// TwinCAT 3 PLC project Untitled1
// ProgramVersion: 3.1.4026.19
// libraries:
//   Tc2_Standard, * (Beckhoff Automation GmbH)
//   Tc2_System, * (Beckhoff Automation GmbH)
// project tree:
//   DUTs/ eGeneralState.TcDUT, eLiftPins.TcDUT, eLiftposition.TcDUT, eLiftStates.TcDUT, eMachineStateLamp.TcDUT, eModus.TcDUT, eSchuifStates.TcDUT, eSingleState.TcDUT, eSlideposition.TcDUT, eStartStop.TcDUT, eValvePosition.TcDUT, eZuigerCilinderposition.TcDUT, eZuigerHorizontaal.TcDUT
//   / PlcTask.TcTTO
//   POUs/ FB_Band.TcPOU, FB_Blinking.TcPOU, FB_ControlSystem.TcPOU, FB_Depalletizer.TcPOU, FB_Lift.TcPOU, FB_LiftA_Extended.TcPOU, FB_LiftB_Extended.TcPOU, FB_LiftJanno.TcPOU, FB_Palletizer.TcPOU, FB_Schuif.TcPOU, FB_Zuiger.TcPOU, FB_Blinking.TcPOU, F_StateEnumToStringSingleState.TcPOU, FB_BlikjesBand.TcPOU, FB_BufferMetKlep.TcPOU, FB_BufferZonderKlep.TcPOU, FB_Invoer.TcPOU, FB_Klep.TcPOU, FB_Simulation.TcPOU, FB_StateManager.TcPOU, GVL.TcGVL, MAIN.TcPOU, F_StateEnumToStringGeneralState.TcPOU
// real-time tasks:
//   TASK PlcTask: cycle T#10ms, priority 20, ADS port 350

CONFIGURATION Untitled1
    RESOURCE PLC ON TwinCAT3
        TASK PlcTask(INTERVAL := T#10ms, PRIORITY := 20);
        PROGRAM MAIN WITH PlcTask : MAIN;
    END_RESOURCE
END_CONFIGURATION

// ---- DUTs/eGeneralState.TcDUT
{attribute 'qualified_only'}
{attribute 'strict'}
{attribute 'to_string'}
TYPE eGeneralState :
(
	Idle 		:= 0,
	Execute		:= 1,
	Stopped 	:= 2,
	Aborted 	:= 3
);
END_TYPE

// ---- DUTs/eLiftPins.TcDUT
{attribute 'qualified_only'}
{attribute 'strict'}
{attribute 'to_string'}
TYPE eLiftPins :
(
	In := 0,
	Out := 1,
	Unknown := 2
);
END_TYPE

// ---- DUTs/eLiftposition.TcDUT
{attribute 'qualified_only'}
{attribute 'strict'}
{attribute 'to_string'}
TYPE eLiftposition :
(
	Idle		:= 0,
	GoingUp 	:= 1,
	GoingDown 	:= 2
	
);
END_TYPE

// ---- DUTs/eLiftStates.TcDUT
{attribute 'qualified_only'}
{attribute 'strict'}
{attribute 'to_string'}
TYPE eLiftStates :
(
	InitHome := 0,
    MoveToHome := 1,
    Impale := 2,
    MoveUpToLayer := 3
);
END_TYPE

// ---- DUTs/eMachineStateLamp.TcDUT
{attribute 'qualified_only'}
{attribute 'strict'}
{attribute 'to_string'}
TYPE eMachineStateLamp :
(
	Green 		:= 0,
	Orange 		:= 1,
	Red			:= 2,
	Red_Blink 	:= 3
	
);
END_TYPE

// ---- DUTs/eModus.TcDUT
{attribute 'qualified_only'}
{attribute 'strict'}
{attribute 'to_string'}
TYPE eModus :
(
	Off := 0,
	Auto := 1,
	Manual := 2
);
END_TYPE

// ---- DUTs/eSchuifStates.TcDUT
{attribute 'qualified_only'}
{attribute 'strict'}
{attribute 'to_string'}
TYPE eSchuifStates :
(
	MoveOut := 0,
	WaitingForConveyor := 1,
	MovingHome := 2,
	Idle := 3
);
END_TYPE

// ---- DUTs/eSingleState.TcDUT
{attribute 'qualified_only'}
{attribute 'strict'}
{attribute 'to_string'}
TYPE eSingleState :
(
	Idle 		:= 0,
	Execute 	:= 1,
	Stopping 	:= 2,
	Stopped 	:= 3,
	Suspending 	:= 4,
	Suspended 	:= 5,
	Aborting 	:= 6,
	Aborted 	:= 7
);
END_TYPE

// ---- DUTs/eSlideposition.TcDUT
{attribute 'qualified_only'}
{attribute 'strict'}
{attribute 'to_string'}
TYPE eSlideposition :
(
	In := 0,
	Out:=1,
	Unknown:=2
);
END_TYPE

// ---- DUTs/eStartStop.TcDUT
{attribute 'qualified_only'}
{attribute 'strict'}
{attribute 'to_string'}
TYPE eStartStop :
(
	Stop 	:= 0,
	Start	:= 1
);
END_TYPE

// ---- DUTs/eValvePosition.TcDUT
{attribute 'qualified_only'}
{attribute 'strict'}
{attribute 'to_string'}
TYPE eValvePosition :
(
	Up := 0,
	Down:=1,
	Unkown:=2
);
END_TYPE

// ---- DUTs/eZuigerCilinderposition.TcDUT
{attribute 'qualified_only'}
{attribute 'strict'}
{attribute 'to_string'}
TYPE eZuigerCilinderposition :
(
	Up := 0,
	Down:=1,
	Unkown:=2
);
END_TYPE

// ---- DUTs/eZuigerHorizontaal.TcDUT
{attribute 'qualified_only'}
{attribute 'strict'}
{attribute 'to_string'}
TYPE eZuigerHorizontaal :
(
	In := 0,
	Out:=1,
	Unkown:=2
);
END_TYPE

// ---- POUs/GVL.TcGVL
{attribute 'qualified_only'}
VAR_GLOBAL
	g_xSimulationActive :BOOL :=TRUE;
	Timerlong : TON;
	TimerShort : TON;
	Timerhmi: TON;
END_VAR

// ---- POUs/MAIN.TcPOU
PROGRAM MAIN
VAR
	//instance of the functionblocks
	fbStateManager					: FB_StateManager;
	fbControlSystem					: FB_ControlSystem;
	fbInvoerBuffer1 				: FB_Invoer;
	fbBuffer2						: FB_BufferZonderKlep;
	fbBuffer3						: FB_BufferZonderKlep;
	fbBuffer4						: FB_BufferZonderKlep;
	fbBuffer5						: FB_BufferMetKlep;
	fbBandDepalletizerPalletizer	: FB_BufferMetKlep;
	fbBlikjesBand					: FB_BlikjesBand;
	fbsim							: FB_Simulation;
	fbDepalletizer					: FB_Depalletizer;
	fbPalletizer					: FB_Palletizer;
	fbSimulation					: FB_Simulation;
	
	//safety
	xAbortGeneral				: BOOL;
	xAbortInvoerBuffer1			: BOOL;
	xAbortPalletizer			: BOOL;
	
	//start stop
	eStartStopGeneral			: eStartStop;
	
	//empty buffers/banden
	xBuffer2Empty						: BOOL;
	xBuffer3Empty						: BOOL;
	xBuffer4Empty						: BOOL;
	xBuffer5Empty						: BOOL;
	xDepalletizerEmpty					: BOOL;
	xBandDepalletizerPalletizerEmpty	: BOOL;
	xPalletizerEmpty					: BOOL;
	
	//buffer/band is emptying
	xInvoerBuffer1Emptying				: BOOL;
	xBuffer2Emptying					: BOOL;
	xBuffer3Emptying					: BOOL;
	xBuffer4Emptying					: BOOL;
	xBuffer5Emptying					: BOOL;
	xDepalletizerEmptying				: BOOL;
	xBandDepalletizerPalletizerEmptying	: BOOL;
	xBlikjesBandAccepting				: BOOL;
	
	// current and next state
	eStateInvoerBuffer1					: eSingleState;
	eStateBuffer2						: eSingleState;
	eStateBuffer3						: eSingleState;
	eStateBuffer4						: eSingleState;
	eStateBuffer5						: eSingleState;
	eStateDepalletizer					: eSingleState;
	eStateBandDepalletizerPalletizer	: eSingleState;
	eStatePalletizer					: eSingleState;
	eStateBlikjesBand					: eSingleState;
	
	//genaral state
	eGeneralState						: eGeneralState;

END_VAR

//----StateManager------------------------------------------------------------------------------------------------------------					
fbStateManager(	i_eStateInvoerBuffer1				:= eStateInvoerBuffer1, 
				i_eStateBuffer2						:= eStateBuffer2, 
				i_eStateBuffer3						:= eStateBuffer3, 
				i_eStateBuffer4						:= eStateBuffer4, 
				i_eStateBuffer5						:= eStateBuffer5, 
				i_eStateDepalletizer				:= eStateDepalletizer, 
				i_eStateBandDepalletizerPalletizer	:= eStateBandDepalletizerPalletizer, 
				i_eStatePalletizer					:= eStatePalletizer, 
				i_eStateBlikjesBand					:= eStateBlikjesBand, 
				o_eGeneralState						=> eGeneralState,
				o_sGeneralStateString				=> );

//----ControlSystem------------------------------------------------------------------------------------------------------------					
fbControlSystem(i_eGeneralState					:= eGeneralState, 
				i_xEmergencyButton				:= (*Used in HMI*), 
				i_xSafetyMat					:= (*Used in HMI*), 
				i_xSafetyDoor					:= (*Used in HMI*), 
				i_xStartButton					:= (*Used in HMI*), 
				i_xStopButton					:= (*Used in HMI*), 
				i_xWarningResetSafetyMat		:= (*Used in HMI*), 
				i_xWarningResetSafetyDoor		:= (*Used in HMI*), 
				i_xAlarmResetPressureGeneral	:= (*Used in HMI*), 
				i_xAlarmResetEmergencyButton	:= (*Used in HMI*), 
				i_iPressureSensorGeneral		:= (*Used in HMI*), 
				o_eStartStopGeneral				=> eStartStopGeneral, 
				o_xWarningSafetyMat				=> (*Used in HMI*), 
				o_xWarningSafetyDoor			=> (*Used in HMI*), 
				o_xAlarmPressureGeneral			=> (*Used in HMI*), 
				o_xAlarmEmergencyButton			=> (*Used in HMI*), 
				o_xErrorPressureGeneral			=> (*Used in HMI*), 
				o_xErrorEmergencyButton			=> (*Used in HMI*), 
				o_xAbortGeneral					=> xAbortGeneral, 
				o_xAbortInvoerBuffer1			=> xAbortInvoerBuffer1, 
				o_xAbortPalletizer				=> xAbortPalletizer, 
				o_eMachineStateLamp1			=> (*Used in HMI*), 
				o_eMachineStateLamp2			=> (*Used in HMI*));
					
//----invoer/buffer 1------------------------------------------------------------------------------------------------------------					
fbInvoerBuffer1(i_xAbort			:= xAbortGeneral OR xAbortInvoerBuffer1, 
				i_eStartStop		:= eStartStopGeneral, 
				i_xPalletPlaced		:= (*Used in HMI*), 
				i_xLightSensor		:= , 
				i_xNextEmpty		:= xBuffer2Empty, 
				i_xAlarmReset		:= (*Used in HMI*), 
				i_eNextState		:= eStateBuffer2,
				i_eModus			:= (*Used in HMI*),
				i_xManualCmdMotor 	:= (*Used in HMI*),	 
				o_eState			=> eStateInvoerBuffer1, 
				o_xMotor			=> (*Used in HMI*), 
				o_xErrorGeneral		=> (*Used in HMI*), 
				o_xAlarmGeneral		=> (*Used in HMI*), 
				o_xGivingToNext		=> xInvoerBuffer1Emptying,
				o_xEmpty			=> (*Used in HMI*),
				o_sStateString		=> (*Used in HMI*));	
				
//----buffer 2------------------------------------------------------------------------------------------------------------							
 fbBuffer2( i_xAbort				:= xAbortGeneral, 
			i_eStartStop			:= eStartStopGeneral,  
			i_xLightSensor			:= ,
			i_xPreviousEmptying	 	:= xInvoerBuffer1Emptying, 
			i_xNextEmpty			:= xBuffer3Empty, 
			i_xAlarmReset			:= (*Used in HMI*), 
			i_eNextState			:= eStateBuffer3, 
			i_eModus				:= (*Used in HMI*),
			i_xManualCmdMotor 		:= (*Used in HMI*),
			o_eState				=> eStateBuffer2, 
			o_xMotor				=> (*Used in HMI*), 
			o_xErrorGeneral			=> (*Used in HMI*), 
			o_xAlarmGeneral			=> (*Used in HMI*), 
			o_xGivingToNext			=> xBuffer2Emptying,
			o_xEmpty 				=> xBuffer2Empty,
			o_sStateString			=> (*Used in HMI*));

//----buffer 3------------------------------------------------------------------------------------------------------------							 
fbBuffer3(  i_xAbort				:= xAbortGeneral, 
			i_eStartStop			:= eStartStopGeneral,  
			i_xLightSensor			:= ,
			i_xPreviousEmptying 	:= xBuffer2Emptying, 
			i_xNextEmpty			:= xBuffer4Empty, 
			i_xAlarmReset			:= (*Used in HMI*), 
			i_eNextState			:= eStateBuffer4, 
			i_eModus				:= (*Used in HMI*),
			i_xManualCmdMotor 		:= (*Used in HMI*),
			o_eState				=> eStateBuffer3, 
			o_xMotor				=> (*Used in HMI*), 
			o_xErrorGeneral			=> (*Used in HMI*), 
			o_xAlarmGeneral			=> (*Used in HMI*), 
			o_xGivingToNext			=> xBuffer3Emptying,
			o_xEmpty 				=> xBuffer3Empty,
			o_sStateString			=> (*Used in HMI*));
			
//----buffer 4------------------------------------------------------------------------------------------------------------							
 fbBuffer4(  i_xAbort				:= xAbortGeneral, 
			i_eStartStop			:= eStartStopGeneral,  
			i_xLightSensor			:= ,
			i_xPreviousEmptying 	:= xBuffer3Emptying, 
			i_xNextEmpty			:= xBuffer5Empty, 
			i_xAlarmReset			:= (*Used in HMI*), 
			i_eNextState			:= eStateBuffer5, 
			i_eModus				:= (*Used in HMI*),
			i_xManualCmdMotor 		:= (*Used in HMI*),
			o_eState				=> eStateBuffer4, 
			o_xMotor				=> (*Used in HMI*), 
			o_xErrorGeneral			=> (*Used in HMI*),
			o_xAlarmGeneral			=> (*Used in HMI*), 
			o_xGivingToNext			=> xBuffer4Emptying,
			o_xEmpty 				=> xBuffer4Empty,
			o_sStateString			=> (*Used in HMI*));

//----buffer 5------------------------------------------------------------------------------------------------------------					
fbBuffer5(	i_xAbort				:= xAbortGeneral, 
			i_eStartStop			:= eStartStopGeneral,  
			i_xLightSensor			:= , 
			i_xPreviousEmptying 	:= xBuffer4Emptying,
			i_xNextEmpty			:= xDepalletizerEmpty, 
			i_xAlarmReset			:= (*Used in HMI*), 
			i_eNextState			:= eStateDepalletizer,
			i_eModus				:= (*Used in HMI*),
			i_xManualCmdMotor 		:= (*Used in HMI*), 
			o_eState				=> eStateBuffer5, 
			o_xMotor				=> (*Used in HMI*), 
			o_xErrorGeneral			=> (*Used in HMI*),
			o_xAlarmGeneral			=> (*Used in HMI*), 
			o_xGivingToNext			=> xBuffer5Emptying,
			o_xEmpty 				=> xBuffer5Empty,
			o_sStateString			=> (*Used in HMI*));
			
//----depalletizer------------------------------------------------------------------------------------------------------------						
fbDepalletizer( i_xAbort			:= xAbortGeneral, 
				i_eStartStop		:= eStartStopGeneral, 
				i_PreviousEmptying	:= xBuffer5Emptying, 
				i_NextEmpty			:= xBandDepalletizerPalletizerEmpty, 
				i_eNextState		:= eStateBandDepalletizerPalletizer, 
				i_iCanType			:= (*Used in HMI*), 
				i_iNumberOfLayersHMI:= (*Used in HMI*), 
				o_eState			=> eStateDepalletizer, 
				o_xEmpty			=> xDepalletizerEmpty, 
				o_xWarningNoProduct	=> (*Used in HMI*), 
				o_aLayerHeights		=> (*??*));
		
//----band depalletizer/palletizer------------------------------------------------------------------------------------------------------------					
fbBandDepalletizerPalletizer(	i_xAbort				:= xAbortGeneral, 
								i_eStartStop			:= eStartStopGeneral,  
								i_xLightSensor			:= , 
								i_xPreviousEmptying 	:= xDepalletizerEmptying,
								i_xNextEmpty			:= xPalletizerEmpty, 
								i_xAlarmReset			:= (*Used in HMI*), 
								i_eNextState			:= eStatePalletizer,
								i_eModus				:= (*Used in HMI*),
								i_xManualCmdMotor 		:= (*Used in HMI*), 
								o_eState				=> eStateBandDepalletizerPalletizer, 
								o_xMotor				=> (*Used in HMI*), 
								o_xErrorGeneral			=> (*Used in HMI*),
								o_xAlarmGeneral			=> (*Used in HMI*), 
								o_xGivingToNext			=> xBandDepalletizerPalletizerEmptying,
								o_xEmpty 				=> xBandDepalletizerPalletizerEmpty,
								o_sStateString			=> (*Used in HMI*));

//----palletizer------------------------------------------------------------------------------------------------------------						
fbPalletizer(	i_xAbort			:= xAbortGeneral, 
				i_eStartStop		:= eStartStopGeneral, 
				i_PreviousEmptying	:= xBandDepalletizerPalletizerEmptying, 
				i_xDoorOpenButton	:= (*Used in HMI*), 
				i_xWarningReset		:= (*Used in HMI*), 
				i_eModus			:= (*Used in HMI*),  
				o_eState			=> eStatePalletizer, 
				o_iStorageCount		=> (*Used in HMI*), 
				o_xWarningFull		=> (*Used in HMI*), 
				o_xExpectingPallet	=> xPalletizerEmpty);

//----blikjesband------------------------------------------------------------------------------------------------------------						
fbBlikjesBand( 	i_xAbort		 		:= xAbortGeneral,
				i_eStartStop 			:= eStartStopGeneral,
				i_eModus				:= (*Used in HMI*), 
				i_xLightSensor 			:= , 
				i_xAlarmReset			:= (*Used in HMI*), 
				i_xManualMotor			:= (*Used in HMI*), 
				o_eState 				=> eStateBlikjesBand,
				o_xMotor 				=> (*Used in HMI*), 
				o_xWarningFull			=> (*Used in HMI*), 
				o_xAcceptingCans		=> xBlikjesBandAccepting);
				
//----simulation------------------------------------------------------------------------------------------------------------						
fbSimulation();

END_PROGRAM

// ---- POUs/FB_StateManager.TcPOU
FUNCTION_BLOCK FB_StateManager
VAR_INPUT
	i_eStateInvoerBuffer1				: eSingleState;
	i_eStateBuffer2						: eSingleState;
	i_eStateBuffer3						: eSingleState;
	i_eStateBuffer4						: eSingleState;
	i_eStateBuffer5						: eSingleState;
	i_eStateDepalletizer				: eSingleState;
	i_eStateBandDepalletizerPalletizer	: eSingleState;
	i_eStatePalletizer					: eSingleState;
	i_eStateBlikjesBand					: eSingleState;
END_VAR
VAR_OUTPUT
	o_eGeneralState 		: eGeneralState;
	o_sGeneralStateString 	: STRING(30);
END_VAR
VAR
END_VAR

//idle
IF i_eStateInvoerBuffer1 = eSingleState.Idle AND
	i_eStateBuffer2 = eSingleState.Idle AND
	i_eStateBuffer3 = eSingleState.Idle AND
	i_eStateBuffer4 = eSingleState.Idle AND
	i_eStateBuffer5 = eSingleState.Idle AND
	i_eStateDepalletizer = eSingleState.Idle AND
	i_eStateBandDepalletizerPalletizer = eSingleState.Idle AND
	i_eStatePalletizer = eSingleState.Idle AND
	i_eStateBlikjesBand = eSingleState.Idle
THEN
	o_eGeneralState := eGeneralState.Idle;
END_IF

//execute
IF i_eStateInvoerBuffer1 = eSingleState.Execute OR
	i_eStateBuffer2 = eSingleState.Execute OR
	i_eStateBuffer3 = eSingleState.Execute OR
	i_eStateBuffer4 = eSingleState.Execute OR
	i_eStateBuffer5 = eSingleState.Execute OR
	i_eStateDepalletizer = eSingleState.Execute OR
	i_eStateBandDepalletizerPalletizer = eSingleState.Execute OR
	i_eStatePalletizer = eSingleState.Execute OR
	i_eStateBlikjesBand = eSingleState.Execute
THEN
	o_eGeneralState := eGeneralState.Execute;
END_IF

//Stopped
IF i_eStateInvoerBuffer1 = eSingleState.Stopped AND
	i_eStateBuffer2 = eSingleState.Stopped AND
	i_eStateBuffer3 = eSingleState.Stopped AND
	i_eStateBuffer4 = eSingleState.Stopped AND
	i_eStateBuffer5 = eSingleState.Stopped AND
	i_eStateDepalletizer = eSingleState.Stopped AND
	i_eStateBandDepalletizerPalletizer = eSingleState.Stopped AND
	i_eStatePalletizer = eSingleState.Stopped AND
	i_eStateBlikjesBand = eSingleState.Stopped
THEN
	o_eGeneralState := eGeneralState.Stopped;
END_IF

//Aborted
IF i_eStateInvoerBuffer1 = eSingleState.Aborted AND
	i_eStateBuffer2 = eSingleState.Aborted AND
	i_eStateBuffer3 = eSingleState.Aborted AND
	i_eStateBuffer4 = eSingleState.Aborted AND
	i_eStateBuffer5 = eSingleState.Aborted AND
	i_eStateDepalletizer = eSingleState.Aborted AND
	i_eStateBandDepalletizerPalletizer = eSingleState.Aborted AND
	i_eStatePalletizer = eSingleState.Aborted AND
	i_eStateBlikjesBand = eSingleState.Aborted
THEN
	o_eGeneralState := eGeneralState.Aborted;
END_IF

//state enum to string for HMI
o_sGeneralStateString := F_StateEnumToStringGeneralState (o_eGeneralState);

END_FUNCTION_BLOCK

// ---- POUs/F_StateEnumToStringGeneralState.TcPOU
FUNCTION F_StateEnumToStringGeneralState : String
VAR_INPUT
		eState  : eGeneralState;
END_VAR
VAR
END_VAR

CASE eState OF
	eGeneralState.Idle:
		F_StateEnumToStringGeneralState := 'Idle';
	eGeneralState.Execute:
		F_StateEnumToStringGeneralState := 'Execute';
	eGeneralState.Stopped:
		F_StateEnumToStringGeneralState := 'Stopped';
	eGeneralState.Aborted:
		F_StateEnumToStringGeneralState := 'Aborted';
ELSE
	F_StateEnumToStringGeneralState := 'Unknown';
END_CASE

END_FUNCTION

// ---- POUs/FB_ControlSystem.TcPOU
FUNCTION_BLOCK FB_ControlSystem
VAR_INPUT
	i_eGeneralState 		: eGeneralState;
	i_xEmergencyButton 		: BOOL;
	i_xSafetyMat 			: BOOL;
	i_xSafetyDoor 			: BOOL;
	i_xStartButton 			: BOOL :=1;
	i_xStopButton 			: BOOL;
	i_xWarningResetSafetyMat			: BOOL;
	i_xWarningResetSafetyDoor			: BOOL;
	i_xAlarmResetPressureGeneral			: BOOL;
	i_xAlarmResetEmergencyButton			: BOOL;
	i_iPressureSensorGeneral: INT := 4000;
	
END_VAR
VAR_OUTPUT
	o_eStartStopGeneral 	: eStartStop;
	
	o_xWarningSafetyMat 	: BOOL;
	o_xWarningSafetyDoor 	: BOOL;
	
	o_xAlarmPressureGeneral	: BOOL;
	o_xAlarmEmergencyButton	: BOOL;
	
	o_xErrorPressureGeneral	: BOOL;
	o_xErrorEmergencyButton	: BOOL;
	
	o_xAbortGeneral			: BOOL;
	o_xAbortInvoerBuffer1	: BOOL;
	o_xAbortPalletizer		: BOOL;
	
	o_eMachineStateLamp1 	: eMachineStateLamp; // Lamp Invoer
	o_eMachineStateLamp2 	: eMachineStateLamp; // Lamp Depalletizer
END_VAR
VAR
	xErrorEmergency			: BOOL := FALSE;
	xErrorPressure			: BOOL := FALSE;
	fbBlinking 				: FB_Blinking;
	
	rlowpressure			: REAL := 4;
	rPressure_bar			: REAL;
	rMaxbarsensor			: REAL :=6;
	
	MachineStateLamp1Blink	: BOOL;
	MachineStateLamp2Blink	: BOOL;
END_VAR

CASE i_eGeneralState OF //read general state and writhes it to the machinestatelamps
	eGeneralState.Aborted:
		o_eMachineStateLamp1 := eMachineStateLamp.Red_Blink;
		o_eMachineStateLamp2 := eMachineStateLamp.Red_Blink;
	eGeneralState.Execute:
		o_eMachineStateLamp1 := eMachineStateLamp.Green;
		o_eMachineStateLamp2 := eMachineStateLamp.Green;
	eGeneralState.Idle:
		o_eMachineStateLamp1 := eMachineStateLamp.Orange;
		o_eMachineStateLamp2 := eMachineStateLamp.Orange;
	eGeneralState.Stopped:
		o_eMachineStateLamp1 := eMachineStateLamp.Red;
		o_eMachineStateLamp2 := eMachineStateLamp.Red;
END_CASE

//blink the machinestatelamps
IF o_eMachineStateLamp1 = eMachineStateLamp.Red_Blink THEN
	fbBlinking(io_xBlinking:= MachineStateLamp1Blink);
END_IF

IF o_eMachineStateLamp2 = eMachineStateLamp.Red_Blink THEN
	fbBlinking(io_xBlinking:= MachineStateLamp2Blink);
END_IF

//safty aborting of machine and parts
IF xErrorEmergency OR xErrorPressure THEN 		 //if emergencybutten or no air pressure then complete machine go's into Aborted
	o_xAbortGeneral := 1;
ELSIF NOT xErrorEmergency AND NOT xErrorPressure THEN
	o_xAbortGeneral := 0;
END_IF
o_xAbortInvoerBuffer1 := i_xSafetyMat; //only for InvoerBuffer 1 Aborted
o_xAbortPalletizer := i_xSafetyDoor; //only of palletizer aborted

//Start Stop
IF i_xStopButton OR  i_eGeneralState=eGeneralState.Aborted THEN //if stopbutton or the machine is aborted the startstop wil become Stop
	o_eStartStopGeneral :=eStartStop.Stop;
	i_xStartButton := FALSE;
END_IF
IF i_xStartButton THEN
	o_eStartStopGeneral :=eStartStop.Start;
	i_xStopButton := FALSE;
END_IF


//pressuresensor error
rPressure_bar := (i_iPressureSensorGeneral / 4095.0) * rMaxbarsensor;// 4095 form analog and 6 from 6 bar max from the sensor
IF rPressure_bar<rlowpressure THEN
	xErrorPressure := TRUE;
ELSE
	xErrorPressure := FALSE;
END_IF

IF xErrorPressure THEN
	fbBlinking(io_xBlinking:= o_xErrorPressureGeneral);
ELSIF NOT xErrorPressure AND o_xAlarmPressureGeneral THEN
	o_xErrorPressureGeneral := TRUE;
ELSE
	o_xErrorPressureGeneral := FALSE;
END_IF;

//Errors
xErrorEmergency := i_xEmergencyButton;

//ALARM
IF xErrorPressure THEN
	o_xAlarmPressureGeneral:=1;
END_IF

IF xErrorEmergency THEN
	o_xAlarmEmergencyButton:=1;
END_IF

//blinking error
IF xErrorEmergency THEN
	fbBlinking(io_xBlinking:= o_xErrorEmergencyButton);
ELSIF NOT xErrorEmergency AND o_xAlarmEmergencyButton THEN
	o_xErrorEmergencyButton := TRUE;
ELSE
	o_xErrorEmergencyButton := FALSE;
END_IF;

//Warning
IF o_xAbortInvoerBuffer1 THEN
	o_xWarningSafetyMat:=1;
ELSIF i_xWarningResetSafetyMat THEN
	o_xWarningSafetyMat:=0;
END_IF

IF o_xAbortPalletizer THEN
	o_xWarningSafetyDoor:=1;
ELSIF i_xWarningResetSafetyDoor THEN
	o_xWarningSafetyDoor:=0;
END_IF

//ERROR reset
IF NOT xErrorPressure AND i_xAlarmResetPressureGeneral THEN
	o_xAlarmPressureGeneral:=0;
END_IF
IF NOT xErrorEmergency AND i_xAlarmResetEmergencyButton THEN
	o_xAlarmEmergencyButton:=0;
END_IF

END_FUNCTION_BLOCK

// ---- POUs/FB_Blinking.TcPOU
FUNCTION_BLOCK FB_Blinking
VAR_IN_OUT
	io_xBlinking		: BOOL;
END_VAR
VAR
	tBlink     		: TON;       
    xBlink     		: BOOL;    
END_VAR

tBlink(IN := TRUE, PT := T#500MS);  

IF tBlink.Q THEN
    xBlink := NOT xBlink;     
    tBlink(IN := FALSE);        
ELSE
    tBlink(IN := TRUE);       
END_IF

io_xBlinking := xBlink;

END_FUNCTION_BLOCK

// ---- POUs/FB_Invoer.TcPOU
FUNCTION_BLOCK FB_Invoer
VAR_INPUT
	i_xAbort		 	: BOOL;
	i_eStartStop 		: eStartStop;
	i_xPalletPlaced		: BOOL := FALSE;			//opperator confirmed that he has placed a pallet
	i_xLightSensor 		: BOOL;
	i_xNextEmpty		: BOOL;
	i_xAlarmReset		: BOOL;
	i_eNextState		: eSingleState;
	i_eModus			: eModus := eModus.Auto;
	i_xManualCmdMotor	: BOOL;
END_VAR
VAR_OUTPUT
	o_eState 			: eSingleState := eSinglestate.Idle;
	o_xMotor 			: BOOL := FALSE;
	o_xErrorGeneral	 	: BOOL := FALSE;
	o_xAlarmGeneral		: BOOL;
	o_xGivingToNext		: BOOL;
	o_xEmpty			: BOOL	:= TRUE;
	o_sStateString 		: STRING(30);
END_VAR
VAR
	xError						 	: BOOL := FALSE;
	tonError						: TON;
	fbBlinking 						: FB_Blinking;
	
	rTrigPallet						: R_TRIG;
	xPalletPresent 					: BOOL;
	tonPalletDetected				: TON;
	xTimerPalletDetectedCompleted 	: BOOL;
	
	fbKlep 							: FB_Klep;
	eValveCurrentPosition			: eValvePosition;
	
	SIMFUNCTIONING: BOOL :=1;
END_VAR

//-------------------------------------------------------------------------------------------------------------------------
//init objects
fbKlep(	i_eState 						:= o_eState,
		i_eModus						:= i_eModus,
		i_eAutoWantedPosition 			:= (*Set in this FB*),
		i_eManualWantedPosition 		:= (*Used in HMI*),
		i_xHallSensorIn 				:= ,
		i_xHallSensorOut 				:= ,
		i_xWarningReset 				:= (*Used in HMI*),
		i_xAlarmReset 					:= (*Used in HMI*),
		o_eCurrentPosition 				=> eValveCurrentPosition,	
		o_xMagnetValve					=> ,
		o_xWarningPositionDown 			=> (*Used in HMI*),
		o_xErrorPositionUpOrUnknow		=> (*Used in HMI*),
		o_xAlarmPositionUpOrUnknow		=> (*Used in HMI*));

//-------------------------------------------------------------------------------------------------------------------------
//Change the state
//execute
IF NOT (i_eModus = eModus.Off) AND (i_eStartStop = eStartStop.Start) AND NOT i_xAbort AND NOT xError THEN
	o_eState := eSingleState.Execute;
END_IF

//stop request
IF i_eStartStop = eStartStop.Stop OR i_eModus = eModus.Off THEN
	o_eState := eSingleState.Stopping;
END_IF

//stopping
IF o_eState = eSingleState.Stopping AND o_xMotor = FALSE THEN
	o_eState := eSingleState.Stopped;
END_IF

//suspening
IF (NOT i_xAbort AND NOT (o_eState = eSingleState.Stopped))  AND 
   (i_eNextState = eSingleState.Suspended OR
    i_eNextState = eSingleState.Stopped   OR
    i_eNextState = eSingleState.Aborted) THEN
	o_eState := eSingleState.Suspending;
END_IF

//suspended
IF o_eState = eSingleState.Suspending AND o_xMotor = FALSE THEN
	o_eState := eSingleState.Suspended;
END_IF

IF i_xAbort THEN
	o_eState := eSingleState.Aborting;
END_IF

//aborted
IF o_eState = eSingleState.Aborting AND o_xMotor = FALSE THEN
	o_eState := eSingleState.aborted;
END_IF

//-----------------------------------------------------------------------------------------------------------------------------------------
//Check error and set error, alarm and state = aboarting
tonError(IN := xPalletPresent AND NOT i_xLightSensor AND o_xMotor, PT := T#20S);
IF  o_xMotor AND tonError.Q THEN
    o_eState := eSingleState.Aborting;
	
	IF tonError.Q THEN
		xError := TRUE;
		o_xAlarmGeneral := TRUE;
	END_IF
END_IF;

//blinking error
IF xError THEN
	fbBlinking(io_xBlinking:= o_xErrorGeneral);
ELSIF NOT xError AND o_xAlarmGeneral THEN
	o_xErrorGeneral := TRUE;
ELSE
	o_xErrorGeneral := FALSE;
END_IF;

//----------------------------------------------------------------------------------------------------------------------------------------
//Trigger the palletplaced value and save in local var
rTrigPallet(CLK := i_xPalletPlaced);
IF rTrigPallet.Q AND NOT xPalletPresent THEN
    xPalletPresent := TRUE;
ELSIF xPalletPresent AND i_xLightSensor AND NOT o_xGivingToNext THEN
	o_xEmpty 		:= FALSE;
ELSIF (xTimerPalletDetectedCompleted AND NOT i_xLightSensor)THEN
	xPalletPresent := FALSE;
	o_xEmpty 	   := TRUE;
	xTimerPalletDetectedCompleted := FALSE; 
END_IF

//----------------------------------------------------------------------------------------------------------------------------------------
//check if pallet detected
tonPalletDetected(IN := i_xLightSensor, PT := T#2S);
IF tonPalletDetected.Q THEN
    xTimerPalletDetectedCompleted := TRUE; 
END_IF

//----------------------------------------------------------------------------------------------------------------------------------------
//motor on
IF 	(i_eModus = eModus.Auto) AND 
	(o_eState = eSingleState.Execute AND xPalletPresent AND NOT i_xLightSensor OR 
	 o_eState = eSingleState.Execute AND i_xLightSensor AND i_xNextEmpty AND eValveCurrentPosition = eValvePosition.Down) OR
	(i_eModus = eModus.Manual AND i_xManualCmdMotor) THEN

	o_xMotor := TRUE;
END_IF

//motor off 
IF  (i_eModus = eModus.Auto) AND 
	(o_eState = eSingleState.Execute AND i_xLightSensor AND NOT i_xNextEmpty OR 
	o_eState = eSingleState.Stopping OR
	o_eState = eSingleState.Suspending OR
	o_eState = eSingleState.Aborting) OR
	(i_eModus = eModus.Manual AND NOT i_xManualCmdMotor) OR
	(NOT xPalletPresent) THEN

	o_xMotor := FALSE;		
END_IF

//----------------------------------------------------------------------------------------------------------------------------------------
//klep position and write o_xGivingToNext
IF o_eState = eSingleState.Execute AND i_xLightSensor AND NOT i_xNextEmpty THEN
	fbKlep(i_eAutoWantedPosition := eValvePosition.Up);
	o_xGivingToNext := FALSE;
	
ELSIF o_eState = eSingleState.Execute AND i_xLightSensor AND i_xNextEmpty THEN
	fbKlep(i_eAutoWantedPosition := eValvePosition.Down);
	IF eValveCurrentPosition = eValvePosition.Down THEN
		 o_xGivingToNext := TRUE;
	END_IF
	
ELSIF NOT i_xLightSensor AND NOT i_xNextEmpty THEN //then placed on the next buffer
	o_xGivingToNext := FALSE;
END_IF

//-------------------------------------------------------------------------------------------------------------------
//reset error
IF NOT (o_eState = eSingleState.Aborting) AND i_xLightSensor THEN
	xError := FALSE;
END_IF

//reset alarm
IF i_xAlarmReset AND NOT xError AND NOT (o_eState = eSingleState.Aborting) THEN
	o_xAlarmGeneral := FALSE;
END_IF

//state enum to string for HMI
o_sStateString := F_StateEnumToStringSingleState(o_eState);


//sim
IF gvl.g_xSimulationActive THEN
	IF SIMFUNCTIONING THEN  
		//
		IF xPalletPresent AND o_xMotor AND gvl.Timerlong.Q AND NOT i_xLightSensor THEN
			i_xLightSensor:=1;
		ELSIF i_xNextEmpty AND o_xMotor AND gvl.Timerlong.Q AND i_xLightSensor THEN
			i_xLightSensor:=0;
		END_IF
	END_IF
END_IF

END_FUNCTION_BLOCK

// ---- POUs/FB_Klep.TcPOU
FUNCTION_BLOCK FB_Klep
VAR_INPUT
	i_eState 				: eSingleState;
	i_eModus				: eModus;
	i_eAutoWantedPosition 	: eValvePosition;
	i_eManualWantedPosition	: eValvePosition;
	i_xHallSensorIn			: BOOL := TRUE;
	i_xHallSensorOut 		: BOOL;
	i_xWarningReset			: BOOL;
	i_xAlarmReset			: BOOL;
END_VAR
VAR_OUTPUT
	o_eCurrentPosition 			: eValvePosition;
	o_xMagnetValve				: BOOL;
	o_xWarningPositionDown 		: BOOL; //Warning when position is down becease it not stopped the machineflow
	o_xErrorPositionUpOrUnknow	: BOOL; //Error when valve is up or unknow beceause it stopped te flow of the machine
	o_xAlarmPositionUpOrUnknow	: BOOL;
END_VAR
VAR
	modeAuto					: BOOL;
	modeManual					: BOOL;
	Timer 						: TON;
	IN 							: BOOL;
	PT 							: TON;
	TimerValue 					: TIME := T#10S;
	TimerStartButton 			: BOOL;
	fbBlinking 					: FB_Blinking;
	xError						: BOOL;
	SIMFUNCTIONING : BOOL := 1;
END_VAR

// Van Emma

// om zetten van enum naar interne bools voor makkelijkheid
CASE i_eModus OF
	eModus.Off:
		modeAuto := FALSE;
		modeManual := FALSE;
	eModus.Auto:
		modeAuto := TRUE;
		modeManual := FALSE;
	eModus.Manual:
		modeAuto := FALSE;
		modeManual := TRUE;
END_CASE 

//stateeeeeee maaaaaacccccchhhhhhiiiiiiinnnnnneeeeee
CASE i_eState OF
	eSingleState.Idle:
		// beneden positie
		GoDown();
	eSingleState.Execute:
		// Ga naar de gewenste stand
		// wanneer auto en manual
		IF modeAuto THEN
			CASE i_eAutoWantedPosition OF
			eValvePosition.Down:
				GoDown();

			eValvePosition.Up:
				GoUp();

			eValvePosition.Unkown:
				TimerStartButton := TRUE;
		
			END_CASE
		ELSIF modeManual THEN
			CASE i_eManualWantedPosition OF
			eValvePosition.Down:
				GoDown();

			eValvePosition.Up:
				GoUp();

			eValvePosition.Unkown:
				TimerStartButton := TRUE;
		
			END_CASE
		END_IF
		
	eSingleState.Stopping:
		// naar beneden
		GoDown();
	eSingleState.Stopped:
		GoDown();
		// niks aansturen alles uit		
	eSingleState.Suspending:
		// Wachten
	eSingleState.Suspended:
		// Wachten
	eSingleState.Aborting:
		// alles uit zetten
		GoDown();
	eSingleState.Aborted:
		GoDown();
END_CASE

// bepaal de huidige positie
IF	i_xHallSensorIn AND i_xHallSensorOut THEN
	o_eCurrentPosition := eValvePosition.Unkown;
ELSIF i_xHallSensorIn	THEN
	o_eCurrentPosition := eValvePosition.Down;
ELSIF i_xHallSensorOut THEN
	o_eCurrentPosition := eValvePosition.Up;
ELSE
	o_eCurrentPosition := eValvePosition.Unkown;
END_IF

// controleer op de klep op de goede positie is 
IF modeAuto AND o_eCurrentPosition = i_eAutoWantedPosition THEN
	xError := FALSE;
	TimerStartButton := FALSE;
ELSIF modeManual AND o_eCurrentPosition = i_eManualWantedPosition THEN
	xError := FALSE;
	TimerStartButton := FALSE;
ELSE 
	TimerStartButton := TRUE;
END_IF

// timer om te kijken of het lang genoeg fout gaat dat het een error is 
Timer(IN:=TimerStartButton, PT := TimerValue);

IF Timer.Q THEN
	Errors(); // method dat als er iets niet goed gaat dat we ook weten wat niet goed gaat
END_IF

// dit is een method om de alarmen te resetten
Resets();

//blinking error van tessa
IF xError THEN
	fbBlinking(io_xBlinking:= o_xErrorPositionUpOrUnknow);
ELSIF NOT xError AND o_xAlarmPositionUpOrUnknow THEN
	o_xErrorPositionUpOrUnknow := TRUE;
ELSE
	o_xErrorPositionUpOrUnknow := FALSE;
END_IF;

//sim van janno
IF gvl.g_xSimulationActive THEN
	IF SIMFUNCTIONING THEN
		IF GVL.TimerShort.Q THEN
			IF o_xMagnetValve THEN
				i_xHallSensorIn :=FALSE;
				i_xHallSensorOut := TRUE;
			ELSE 
				i_xHallSensorOut := FALSE;
				i_xHallSensorIn :=TRUE;
			END_IF
		END_IF
	END_IF
END_IF

METHOD Errors
VAR
END_VAR
// als er op de verwachte positie te lang niet iets is dan gaan we hiernaar toe om te kijken wat de error is 

CASE o_eCurrentPosition OF
	eValvePosition.Up :
			xError := TRUE;
			o_xAlarmPositionUpOrUnknow := TRUE;	
	eValvePosition.Down :
			o_xWarningPositionDown := TRUE;
	eValvePosition.Unkown :
			xError := TRUE;
			o_xAlarmPositionUpOrUnknow := TRUE;	
END_CASE
END_METHOD

METHOD GoDown
o_xMagnetValve := FALSE;

// bedenen is magnet valve false
END_METHOD

METHOD GoUp
o_xMagnetValve := TRUE;

// boven is magner valve true
END_METHOD

METHOD Resets
IF 	i_xWarningReset THEN
	o_xWarningPositionDown := FALSE;
	TimerStartButton := FALSE;
END_IF

IF i_xAlarmReset THEN
	TimerStartButton := FALSE;
	o_xAlarmPositionUpOrUnknow := FALSE;
END_IF

// dit is om de alarm en waarschuwing weg te doen
END_METHOD

END_FUNCTION_BLOCK

// ---- POUs/F_StateEnumToStringSingleState.TcPOU
FUNCTION F_StateEnumToStringSingleState : STRING
VAR_INPUT
	eState  : eSingleState;
END_VAR
VAR
END_VAR

CASE eState OF
	eSingleState.Idle:
		F_StateEnumToStringSingleState := 'Idle';
	eSingleState.Execute:
		F_StateEnumToStringSingleState := 'Execute';
	eSingleState.Stopping:
		F_StateEnumToStringSingleState := 'Stopping';
	eSingleState.Stopped:
		F_StateEnumToStringSingleState := 'Stopped';
	eSingleState.Suspending:
		F_StateEnumToStringSingleState := 'Suspending';
	eSingleState.Suspended:
		F_StateEnumToStringSingleState := 'Suspended';
	eSingleState.Aborting:
		F_StateEnumToStringSingleState := 'Aborting';
	eSingleState.Aborted:
		F_StateEnumToStringSingleState := 'Aborted';
ELSE
	F_StateEnumToStringSingleState := 'Unknown';
END_CASE

END_FUNCTION

// ---- POUs/FB_BufferZonderKlep.TcPOU
FUNCTION_BLOCK FB_BufferZonderKlep
VAR_INPUT
	i_xAbort		 	: BOOL;
	i_eStartStop 		: eStartStop;
	i_xLightSensor 		: BOOL;
	i_xNextEmpty		: BOOL;
	i_xPreviousEmptying	: BOOL;
	i_xAlarmReset		: BOOL;
	i_eNextState		: eSingleState;
	i_eModus			: eModus := eModus.Auto;
	i_xManualCmdMotor	: BOOL;
END_VAR
VAR_OUTPUT
	o_eState 			: eSingleState := eSinglestate.Idle;
	o_xMotor 			: BOOL := FALSE;
	o_xErrorGeneral 	: BOOL := FALSE;
	o_xAlarmGeneral		: BOOL;
	o_xGivingToNext		: BOOL;
	o_xEmpty			: BOOL	:= TRUE;
	o_sStateString 		: STRING(30);
END_VAR
VAR	
	xError				: BOOL;
	tonError			: TON;
	fbBlinking 			: FB_Blinking;
	SIMFUNCTIONING: BOOL :=1;
END_VAR

//-------------------------------------------------------------------------------------------------------------------------
//Change the state
//execute
IF NOT (i_eModus = eModus.Off) AND (i_eStartStop = eStartStop.Start) AND NOT i_xAbort AND NOT xError THEN
	o_eState := eSingleState.Execute;
END_IF

//stop request
IF i_eStartStop = eStartStop.Stop THEN
	o_eState := eSingleState.Stopping;
END_IF

//stopping
IF o_eState = eSingleState.Stopping AND o_xMotor = FALSE THEN
	o_eState := eSingleState.Stopped;
END_IF

//suspening
IF (NOT i_xAbort AND NOT (o_eState = eSingleState.Stopped))  AND 
   (i_eNextState = eSingleState.Suspended OR
    i_eNextState = eSingleState.Stopped   OR
    i_eNextState = eSingleState.Aborted) THEN
	o_eState := eSingleState.Suspending;
END_IF

//suspended
IF o_eState = eSingleState.Suspending AND o_xMotor = FALSE THEN
	o_eState := eSingleState.Suspended;
END_IF

IF i_xAbort THEN
	o_eState := eSingleState.Aborting;
END_IF

//aborted
IF o_eState = eSingleState.Aborting AND o_xMotor = FALSE THEN
	o_eState := eSingleState.aborted;
END_IF

//-----------------------------------------------------------------------------------------------------------------------------------------
//Check error and set error, alarm and state = aboarting
tonError(IN := NOT i_xLightSensor AND o_xMotor, PT := T#20S);
IF  o_xMotor AND tonError.Q THEN
    o_eState := eSingleState.Aborting;
	
	IF tonError.Q THEN
		xError := TRUE;
		o_xAlarmGeneral := TRUE;
	END_IF
END_IF;

//blinking error
IF xError THEN
	fbBlinking(io_xBlinking:= o_xErrorGeneral);
ELSIF NOT xError AND o_xAlarmGeneral THEN
	o_xErrorGeneral := TRUE;
ELSE
	o_xErrorGeneral := FALSE;
END_IF;

//----------------------------------------------------------------------------------------------------------------------------------------
//motor on
IF (i_eModus = eModus.Auto) AND 
	(o_eState = eSingleState.Execute AND i_xPreviousEmptying AND NOT i_xLightSensor OR 
	o_eState = eSingleState.Execute AND i_xLightSensor AND i_xNextEmpty) OR
	(i_eModus = eModus.Manual AND i_xManualCmdMotor) THEN

	o_xMotor := TRUE;
END_IF

//motor off 
IF (i_eModus = eModus.Auto) AND 
	(o_eState = eSingleState.Execute AND i_xLightSensor AND NOT i_xNextEmpty OR 
	o_eState = eSingleState.Stopping OR
	o_eState = eSingleState.Suspending OR
	o_eState = eSingleState.Aborting) OR
	(i_eModus = eModus.Manual AND NOT i_xManualCmdMotor) OR
 	(o_xEmpty AND NOT i_xPreviousEmptying AND NOT (i_eModus = eModus.Manual)) THEN

	o_xMotor := FALSE;		
END_IF

//----------------------------------------------------------------------------------------------------------------------------------------
//write o_xGivingToNext
IF o_eState = eSingleState.Execute AND i_xLightSensor AND NOT i_xNextEmpty THEN
	o_xGivingToNext := FALSE;	
ELSIF o_eState = eSingleState.Execute AND i_xLightSensor AND i_xNextEmpty THEN
	o_xGivingToNext := TRUE;
ELSIF NOT i_xLightSensor AND NOT i_xNextEmpty THEN //then placed on the next buffer
	o_xGivingToNext := FALSE;
END_IF

//----------------------------------------------------------------------------------------------------------------------------------------
//check if buffer is empty
IF NOT i_xLightSensor THEN
	o_xEmpty := TRUE;
ELSE
	o_xEmpty := FALSE;
END_IF

//-------------------------------------------------------------------------------------------------------------------
//reset alarm and error
IF NOT (o_eState = eSingleState.Aborting) AND i_xLightSensor THEN
	xError := FALSE;
END_IF

//reset alarm
IF i_xAlarmReset AND NOT xError AND NOT (o_eState = eSingleState.Aborting) THEN
	o_xAlarmGeneral := FALSE;
END_IF

//state enum to string for HMI
o_sStateString := F_StateEnumToStringSingleState(o_eState);

//sim
IF gvl.g_xSimulationActive THEN
	IF SIMFUNCTIONING THEN 
		IF i_xPreviousEmptying AND o_xMotor AND gvl.Timerlong.Q AND NOT i_xLightSensor THEN
			i_xLightSensor:=1;
		ELSIF i_xNextEmpty AND o_xMotor AND gvl.Timerlong.Q AND i_xLightSensor THEN
			i_xLightSensor:=0;
		END_IF
	END_IF
END_IF

END_FUNCTION_BLOCK

// ---- POUs/FB_BufferMetKlep.TcPOU
FUNCTION_BLOCK FB_BufferMetKlep
VAR_INPUT
	i_xAbort		 	: BOOL;
	i_eStartStop 		: eStartStop;
	i_xLightSensor 		: BOOL;
	i_xNextEmpty		: BOOL;
	i_xPreviousEmptying	: BOOL;
	i_xAlarmReset		: BOOL;
	i_eNextState		: eSingleState;
	i_eModus			: eModus := eModus.Auto;
	i_xManualCmdMotor	: BOOL;
END_VAR
VAR_OUTPUT
	o_eState 			: eSingleState := eSinglestate.Idle;
	o_xMotor 			: BOOL := FALSE;
	o_xErrorGeneral 	: BOOL := FALSE;
	o_xAlarmGeneral		: BOOL;
	o_xGivingToNext		: BOOL;
	o_xEmpty			: BOOL	:= TRUE;
	o_sStateString 		: STRING(30);
END_VAR
VAR
	xError					: BOOL;
	tonError	 			: TON;
	fbBlinking 				: FB_Blinking;
	
	fbKlep 					: FB_Klep;
	eValveCurrentPosition	: eValvePosition;
	SIMFUNCTIONING: BOOL :=1;
END_VAR

//-------------------------------------------------------------------------------------------------------------------------
//init objects
fbKlep(	i_eState 						:= o_eState,
		i_eModus						:= i_eModus,
		i_eAutoWantedPosition 			:= (*Set in this FB*),
		i_eManualWantedPosition 		:= (*Used in HMI*),
		i_xHallSensorIn 				:= ,
		i_xHallSensorOut 				:= ,
		i_xWarningReset 				:= (*Used in HMI*),
		i_xAlarmReset 					:= (*Used in HMI*),
		o_eCurrentPosition 				=> eValveCurrentPosition,	
		o_xMagnetValve					=> ,
		o_xWarningPositionDown 			=> (*Used in HMI*),
		o_xErrorPositionUpOrUnknow		=> (*Used in HMI*),
		o_xAlarmPositionUpOrUnknow		=> (*Used in HMI*));

//-------------------------------------------------------------------------------------------------------------------------
//Change the state
//execute
IF NOT (i_eModus = eModus.Off) AND (i_eStartStop = eStartStop.Start) AND NOT i_xAbort AND NOT xError THEN
	o_eState := eSingleState.Execute;
END_IF

//stop request
IF i_eStartStop = eStartStop.Stop THEN
	o_eState := eSingleState.Stopping;
END_IF

//stopping
IF o_eState = eSingleState.Stopping AND o_xMotor = FALSE THEN
	o_eState := eSingleState.Stopped;
END_IF

//suspening
IF (NOT i_xAbort AND NOT (o_eState = eSingleState.Stopped))  AND 
   (i_eNextState = eSingleState.Suspended OR
    i_eNextState = eSingleState.Stopped   OR
    i_eNextState = eSingleState.Aborted) THEN
	o_eState := eSingleState.Suspending;
END_IF

//suspended
IF o_eState = eSingleState.Suspending AND o_xMotor = FALSE THEN
	o_eState := eSingleState.Suspended;
END_IF

IF i_xAbort THEN
	o_eState := eSingleState.Aborting;
END_IF

//aborted
IF o_eState = eSingleState.Aborting AND o_xMotor = FALSE THEN
	o_eState := eSingleState.aborted;
END_IF

//-----------------------------------------------------------------------------------------------------------------------------------------
//Check error and set error, alarm and state = aboarting
tonError(IN := NOT i_xLightSensor AND o_xMotor, PT := T#20S);
IF  o_xMotor AND tonError.Q THEN
    o_eState := eSingleState.Aborting;
	
	IF tonError.Q THEN
		xError := TRUE;
		o_xAlarmGeneral := TRUE;
	END_IF
END_IF;

//blinking error
IF xError THEN
	fbBlinking(io_xBlinking:= o_xErrorGeneral);
ELSIF NOT xError AND o_xAlarmGeneral THEN
	o_xErrorGeneral := TRUE;
ELSE
	o_xErrorGeneral := FALSE;
END_IF;

//----------------------------------------------------------------------------------------------------------------------------------------
//motor on
IF (i_eModus = eModus.Auto) AND 
	(o_eState = eSingleState.Execute AND i_xPreviousEmptying AND NOT i_xLightSensor OR 
	o_eState = eSingleState.Execute AND i_xLightSensor AND i_xNextEmpty AND eValveCurrentPosition = eValvePosition.Down) OR
	(i_eModus = eModus.Manual AND i_xManualCmdMotor) THEN

	o_xMotor := TRUE;
END_IF

//motor off 
IF (i_eModus = eModus.Auto) AND 
	(o_eState = eSingleState.Execute AND i_xLightSensor AND NOT i_xNextEmpty OR 
	o_eState = eSingleState.Stopping OR
	o_eState = eSingleState.Suspending OR
	o_eState = eSingleState.Aborting) OR
	(i_eModus = eModus.Manual AND NOT i_xManualCmdMotor) OR 
	(o_xEmpty AND NOT i_xPreviousEmptying AND NOT (i_eModus = eModus.Manual)) OR
	NOT(eValveCurrentPosition = eValvePosition.Down) THEN

	o_xMotor := FALSE;		
END_IF

//----------------------------------------------------------------------------------------------------------------------------------------
//klep position and write o_xGivingToNext
IF o_eState = eSingleState.Execute AND i_xLightSensor AND NOT i_xNextEmpty THEN
	fbKlep(i_eAutoWantedPosition 		:= eValvePosition.Up);
	o_xGivingToNext := FALSE;
ELSIF o_eState = eSingleState.Execute AND i_xLightSensor AND i_xNextEmpty THEN
	fbKlep(i_eAutoWantedPosition := eValvePosition.Down);
	IF fbKlep.o_eCurrentPosition = eValvePosition.Down THEN
		o_xGivingToNext := TRUE;
	END_IF
ELSIF NOT i_xLightSensor AND NOT i_xNextEmpty THEN //then placed on the next buffer
	o_xGivingToNext := FALSE;
END_IF

//----------------------------------------------------------------------------------------------------------------------------------------
//check if buffer is empty
IF NOT i_xLightSensor THEN
	o_xEmpty := TRUE;
ELSE
	o_xEmpty := FALSE;
END_IF

//-------------------------------------------------------------------------------------------------------------------
//reset alarm and error
IF NOT (o_eState = eSingleState.Aborting) AND i_xLightSensor THEN
	xError := FALSE;
END_IF

//reset alarm
IF i_xAlarmReset AND NOT xError AND NOT (o_eState = eSingleState.Aborting) THEN
	o_xAlarmGeneral := FALSE;
END_IF

//state enum to string for HMI
o_sStateString := F_StateEnumToStringSingleState(o_eState);

//sim
IF gvl.g_xSimulationActive THEN
	IF SIMFUNCTIONING THEN 
		IF i_xPreviousEmptying AND o_xMotor AND gvl.Timerlong.Q AND NOT i_xLightSensor THEN
			i_xLightSensor:=1;
		ELSIF o_xGivingToNext AND o_xMotor AND gvl.Timerlong.Q AND i_xLightSensor THEN
			i_xLightSensor:=0;
		END_IF
	END_IF
END_IF

END_FUNCTION_BLOCK

// ---- POUs/FB_BlikjesBand.TcPOU
FUNCTION_BLOCK FB_BlikjesBand
VAR_INPUT
	i_xAbort		 		: BOOL;
	i_eStartStop 			: eStartStop;
	i_eModus				: eModus := eModus.Auto; // 0= off 1= auto 2= manual
	i_xLightSensor 			: BOOL; // checking for cans after 10 sec alarm
	i_xAlarmReset			: BOOL;
	i_xManualMotor			: BOOL;
END_VAR
VAR_OUTPUT
	o_eState 				: eSingleState := eSingleState.Idle;
	o_xMotor 				: BOOL := FALSE;
	o_xWarningFull			: BOOL;
	o_xAcceptingCans		: BOOL; //For other machines that this one is working and has space for cans
	o_sStateString 			: STRING(30);
END_VAR
VAR
	xError : BOOL;

	Timer : TON;
	IN : BOOL;
	PT : TON;
	TimerValue : TIME := T#20S;
	TimerStartButton : BOOL;
	SIMFUNCTIONING : BOOL := 1;
END_VAR

// Van Emma

// bijwerken van inner state door de methode aan te roepen
StateChange();

// check modus en doe wat je in de mode moet doen
CASE i_eModus OF
	eModus.Off:
		o_xMotor := FALSE;
		
	eModus.Auto: // als auto is moet ie aan, want hij blijft eigenlijk aan
		o_xMotor := TRUE;
		
	eModus.Manual:
		IF i_xManualMotor THEN
			o_xMotor := TRUE;
		ELSE
			o_xMotor := FALSE;
		END_IF
		
END_CASE

// als lichtsensor true is betekend het dat er te veel bliken op de band zijn
IF i_xLightSensor THEN
	TimerStartButton := TRUE;
END_IF

// timer voor de zekerheid dat er echt te veel zijn en niet eentje die net voor de sensor was
Timer(IN:=TimerStartButton, PT := TimerValue);
IF Timer.Q THEN
	o_xAcceptingCans := FALSE;
	o_xWarningFull := TRUE;
ELSE
	o_xAcceptingCans := TRUE;
END_IF

// arlam reset
IF i_xAlarmReset = TRUE THEN
	TimerStartButton := FALSE;
	o_xWarningFull := FALSE;
END_IF

//state enum to string for HMI
o_sStateString := F_StateEnumToStringSingleState(o_eState);

//sim van janno
IF gvl.g_xSimulationActive THEN
	IF SIMFUNCTIONING THEN
		IF GVL.TimerShort.Q THEN
			i_xLightSensor :=FALSE;
		END_IF
	ELSE
		i_xLightSensor :=TRUE;
	END_IF
END_IF

METHOD StateChange
//execute
IF NOT (i_eModus = eModus.Off) AND (i_eStartStop = eStartStop.Start) AND NOT i_xAbort AND NOT xError THEN
	o_eState := eSingleState.Execute;
END_IF

//stop request
IF i_eStartStop = eStartStop.Stop OR i_eModus = eModus.Off THEN
	o_eState := eSingleState.Stopping;
END_IF

//stopping
IF o_eState = eSingleState.Stopping AND o_xMotor = FALSE THEN
	o_eState := eSingleState.Stopped;
END_IF

//suspening
IF (NOT i_xAbort AND NOT (o_eState = eSingleState.Stopped)) THEN
	o_eState := eSingleState.Suspending;
END_IF

//suspended
IF o_eState = eSingleState.Suspending AND o_xMotor = FALSE THEN
	o_eState := eSingleState.Suspended;
END_IF

IF i_xAbort THEN
	o_eState := eSingleState.Aborting;
END_IF

//aborted
IF o_eState = eSingleState.Aborting AND o_xMotor = FALSE THEN
	o_eState := eSingleState.aborted;
END_IF
END_METHOD

END_FUNCTION_BLOCK

// ---- POUs/FB_Simulation.TcPOU
FUNCTION_BLOCK FB_Simulation
VAR_INPUT
	
END_VAR
VAR_OUTPUT

END_VAR
VAR
	//timers
	timTimerValueLong : TIME := T#7S;
	xTimerLongRunning: BOOL;

	timTimerValueShort : TIME := T#2S;
	xTimerShortRunning: BOOL;
	xTimerhmiRunning: BOOL;
	timTimerValuehmi: TIME := T#20MS;
END_VAR

//timer long and short for simulating wait time before somnething happens in the code
GVL.Timerlong(IN:=xTimerLongRunning, PT:=timTimerValueLong);
IF GVL.Timerlong.Q THEN
	xTimerLongRunning:=FALSE;
ELSE
	xTimerLongRunning:=TRUE;
END_IF

GVL.TimerShort(IN:=xTimerShortRunning, PT:=timTimerValueShort);
IF GVL.TimerShort.Q THEN
	xTimerShortRunning:=FALSE;
ELSE
	xTimerShortRunning:=TRUE;
END_IF

GVL.Timerhmi(IN:=xTimerhmiRunning, PT:=timTimerValuehmi);
IF GVL.Timerhmi.Q THEN
	xTimerhmiRunning:=FALSE;
ELSE
	xTimerhmiRunning:=TRUE;
END_IF

END_FUNCTION_BLOCK

// ---- POUs/FB_Depalletizer.TcPOU
FUNCTION_BLOCK FB_Depalletizer
VAR_INPUT
	i_xAbort		 	: BOOL;														// MOET NOG IETS MEE
	i_eStartStop 		: eStartStop;												// MOET NOG IETS MEE
	i_PreviousEmptying	: BOOL;														// MOET NOG IETS MEE
	i_NextEmpty			: BOOL;
	i_eNextState		: eSingleState;												// MOET NOG IETS MEE
	
	i_HeightSensor		: BOOL;
	
	// HMI
	i_iCanTypeHMI		: INT;	// Type of can loaded on pallet
	i_iNumberOfLayersHMI: INT;	// Number of layers on the pallet
END_VAR
VAR_OUTPUT
	o_eState 			: eSingleState;
	o_xEmpty			: BOOL;	// Depalletizer is empty
	o_xWarningNoProduct	: BOOL; // Warning after ...  time no products detected.
	o_xGivingToNext		: BOOL; // Let the next conveyor know it is getting a new pallet.
	
	o_aLayerHeights	: ARRAY[1..10] OF INT;
END_VAR
VAR
	fbBand: FB_Band;
	fbSchuif: FB_Schuif;
	fbZuiger: FB_Zuiger;
	fbKlep: FB_Klep;
	fbLiftA: FB_LiftA_Extended;
	
	xLiftIsDone		: BOOL;
	xReleasePallet	: BOOL;
	xHoldPallet		: BOOL;
	
	iLayerHeight	: INT;
	iBaseHeight		: INT := 0;
	i				: INT := 0;
	iSlideHeight	: INT := 2500;
	
	eMoveKlep		: eValvePosition;
	
	eCheckZuigerSafe		: eZuigerCilinderPosition;
	eSchuifSafe		: eSlideposition;
	eConveyorSafe	: eValvePosition;
	
	xMoveUpSafe		: BOOL;
	xMoveDownSafe	: BOOL;
	
		// Light Sensors
	xLightSensor1		: BOOL; // De eerste sensor die de pallet detecteerd
	xLightSensor2		: BOOL; // De tweede sensor die de pallet detecteerd
	
	xPalletInPosition	: BOOL;
	
	xConveyorMoving		: BOOL;
	
	xGoZuiger	: BOOL;
	xGoSchuif	: BOOL;
END_VAR

// Yvo

// Check the type of can and give the height of each layer
THIS^.CheckCanType();

// Calculate the layer heights
THIS^.CalculateLayerHeights();

// Set as empty if no sensor detects pallet
THIS^.SetEmpty();

// If sensor detects new pallet, move Klep up
THIS^.DetectNewPallet();

// Check Zuiger and Schuif are safe so the lift can move up
THIS^.CheckMoveUp();

// Check if lift can move down
THIS^.CheckMoveDown();

// If Lift is done, release pallet. If not possible, hold pallet.
THIS^.ReleaseOrHoldPallet();

// Functionblock Klep
fbKlep(
	i_eState:= , 
	i_eModus:= , 
	i_eAutoWantedPosition:= eMoveKlep, 
	i_eManualWantedPosition:= , 
	i_xHallSensorIn:= , 
	i_xHallSensorOut:= , 
	i_xWarningReset:= , 
	i_xAlarmReset:= , 
	o_eCurrentPosition=> , 
	o_xMagnetValve=> , 
	o_xWarningPositionDown=> , 
	o_xErrorPositionUpOrUnknow=> , 
	o_xAlarmPositionUpOrUnknow=> );

// Functionblock Schuif
fbSchuif(
	i_eState:= , 
	i_eMode:= , 
	i_xMove:= xGoSchuif, 
	i_xMovePossible:= , 
	i_xMoveHome:= , 
	i_xEndSwitchIn:= , 
	i_xEndSwitchOut:= , 
	i_xAlarmReset:= , 
	i_xHMIMoveIn:= , 
	i_xHMIMoveOut:= , 
	i_xHMIStopMoving:= , 
	o_xMotor=> , 
	o_xMotorDirection=> , 
	o_xErrorSlide=> , 
	o_xAlarmSlide=> , 
	o_xMoveDone=> , 
	o_eSlidePosition=> );
	
// Functionblock Zuiger
fbZuiger(
	i_eState:= , 
	i_eModes:= , 
	i_xMoveCiliderDown:= , 
	i_xHallSensorIn:= , 
	i_xHallSensorOut:= , 
	i_xEndSwitchIn:= , 
	i_xEndSwitchOut:= , 
	i_rPressureSensor:= , 
	i_xAlarmResetCilinder:= , 
	i_xAlarmResetAlarmHorizontalMovement:= , 
	i_xAlarmResetPressure:= , 
	i_xButtonManStopall:= , 
	eManCiliderPosition:= , 
	eManHorizotalPosition:= , 
	i_xButtonManVacumOn:= , 
	o_xMotor=> , 
	o_xMotorDirectionOut=> , 
	o_xErrorHorizontalMovement=> , 
	o_xAlarmHorizontalMovement=> , 
	o_xMagnetValveCilinder=> , 
	o_xMagnetValveVacum=> , 
	o_xErrorCilinder=> , 
	o_xAlarmCilinder=> , 
	o_xErrorPressure=> , 
	o_xAlarmPressure=> , 
	o_eCiliderPosition=> eCheckZuigerSafe, 
	o_eHorizotalPosition=> );

// Functionblock Lift
fbBand(
	i_eState:= , 
	i_xGoHold:= xHoldPallet, 
	i_xGoEmpty:= xReleasePallet, 
	i_xAlarmReset:= , 
	i_eModus:= , 
	i_xManualMotor:= , 
	o_xMotor=> xConveyorMoving, 
	o_xErrorMotor=> , 
	o_xAlarmMotor=> , 
	o_xGivingToNext=> );
	
// Functionblock Lift
fbLiftA(
	i_eLiftState:= , 
	i_iServoEncoder:= , 
	i_xEndSwitch:= , 
	i_xPin1HallSensorIn:= , 
	i_xPin2HallSensorIn:= , 
	i_xPin3HallSensorIn:= , 
	i_xPin4HallSensorIn:= , 
	i_xPin1HallSensorOut:= , 
	i_xPin2HallSensorOut:= , 
	i_xPin3HallSensorOut:= , 
	i_xPin4HallSensorOut:= , 
	i_xLightSensor1:= xLightSensor1, 
	i_xLightSensor2:= xLightSensor2, 
	i_xMoveUpSafe:= xMoveUpSafe,
	i_xMoveDownSafe:= xMoveDownSafe,
	i_xPalletInPosition:= xPalletInPosition,
	o_iTargetPos=> , 
	o_eLiftPosition=> , 
	o_xMotor=> , 
	o_xMagnetValve=> , 
	o_ePinsPositions=> , 
	i_aLayerHeights:= o_aLayerHeights, 
	i_iLayerCount:= i_iNumberOfLayersHMI, 
	i_xMoveUpSafe:= xMoveUpSafe, 
	i_eZuigerDone:= eCheckZuigerSafe,
	o_xGoSchuif=> xGoSchuif, 
	o_xGoZuiger=> xGoZuiger,
	o_xLiftDone=> xLiftIsDone);

METHOD CalculateLayerHeights : BOOL
VAR_INPUT
END_VAR
FOR i := 1 TO i_iNumberOfLayersHMI DO
	o_aLayerHeights[i] := (iBaseHeight + (i - 1) * iLayerHeight) + (iSlideHeight - iLayerHeight);
END_FOR
END_METHOD

METHOD CheckCanType : BOOL
VAR_INPUT
END_VAR
IF i_iCanTypeHMI = 1 THEN
	iLayerHeight := 500;
ELSIF i_iCanTypeHMI = 2 THEN
	iLayerHeight := 1000;
ELSIF i_iCanTypeHMI = 3 THEN
	iLayerHeight := 1500;
END_IF
END_METHOD

METHOD CheckMoveDown : BOOL
VAR_INPUT
END_VAR
IF eConveyorSafe = eValvePosition.Down THEN
	xMoveDownSafe := TRUE;
ELSE
	xMoveDownSafe := FALSE;
END_IF
END_METHOD

METHOD CheckMoveUp : BOOL
VAR_INPUT
END_VAR
IF eCheckZuigerSafe = eZuigerCilinderPosition.Up AND eSchuifSafe = eSlidePosition.In THEN
	xMoveUpSafe := TRUE;
ELSE
	xMoveUpSafe := FALSE;
END_IF
END_METHOD

METHOD DetectNewPallet : BOOL
(*
	This Method detects a new pallet on the conveyor.
	When the first sensor detects a pallet, Klep will be moved up to stop the pallet from going to far.
	When Sensor 2 also detects the pallet, the conveyor will be told to stop moving.
	When the conveyor stops moving, the klep will be moved down and the signal "pallet in position" will be send to the lift.
*)
VAR_INPUT
END_VAR
IF xLightSensor1 THEN
	// Move klep up
	eMoveKlep := eValvePosition.Up;
	xHoldPallet := FALSE;
	xPalletInPosition := FALSE;
	IF xLightSensor2 THEN
		xHoldPallet := TRUE;
		IF xConveyorMoving = FALSE THEN
			eMoveKlep := eValvePosition.Down;
			IF eMoveKlep = eValvePosition.Down THEN
				xPalletInPosition := TRUE;
			END_IF
		END_IF
	ELSE
		xHoldPallet := FALSE;
		xPalletInPosition := FALSE;
	END_IF
END_IF
END_METHOD

METHOD ReleaseOrHoldPallet : BOOL
VAR_INPUT
END_VAR
IF xLiftIsDone AND i_NextEmpty THEN
	xReleasePallet := TRUE;
	xHoldPallet := FALSE;
	o_xGivingToNext := TRUE;
ELSIF xLiftIsDone AND i_NextEmpty = FALSE THEN
	xHoldPallet := TRUE;
	xReleasePallet := FALSE;
END_IF
END_METHOD

METHOD SetEmpty : BOOL
VAR_INPUT
END_VAR
IF xLightSensor1 = FALSE AND xLightSensor2 = FALSE THEN
	o_xEmpty := TRUE;
ELSE 
	o_xEmpty := FALSE;
END_IF
END_METHOD

END_FUNCTION_BLOCK

// ---- POUs/FB_Band.TcPOU
FUNCTION_BLOCK FB_Band
VAR_INPUT
	i_eState		: eSingleState;
	i_xGoHold 		: BOOL; //keep pallet on band wachten
	i_xGoEmpty		: BOOL; //move pallet to other segment go
	i_xAlarmReset	: BOOL;
	i_eModus		: eModus := eModus.Auto;
	i_xManualMotor  : BOOL;
END_VAR
VAR_OUTPUT
	o_xMotor 		: BOOL := FALSE;
	o_xErrorMotor 	: BOOL := FALSE;
	o_xAlarmMotor	: BOOL;
	o_xGivingToNext	: BOOL;
END_VAR
VAR
	fbBlinking : FB_Blinking;
	xError : Bool;
END_VAR

// Van Emma :)

CASE i_eModus OF
	eModus.Off: 
		o_xMotor := FALSE;
		
	eModus.Auto:
		IF i_xGoHold = TRUE THEN
			o_xMotor := FALSE; // go hold betekend dat de pallet moet blijven dus motor uit
		ELSIF i_xGoEmpty = TRUE THEN
			o_xMotor := TRUE; // go empty betekend dat de pallet weg moet dus motor aan
			o_xGivingToNext := TRUE;
		ELSE
			o_xGivingToNext := FALSE;
		END_IF
		
		// error logica dit genereert een fout als de motor aan staat terwijl die uit moet zijn
		IF i_xGoEmpty = FALSE AND o_xMotor = TRUE THEN
			xError := TRUE;	
			o_xAlarmMotor := TRUE;
		ELSIF i_xGoHold = TRUE AND o_xMotor = TRUE THEN
			xError := TRUE;	
			o_xAlarmMotor := TRUE;
		ELSE
			xError := FALSE;	
		END_IF 
		
	eModus.Manual:
		IF i_xManualMotor THEN
			o_xMotor := TRUE;
		ELSE
			o_xMotor := FALSE;
		END_IF
		
END_CASE



// alarm reset
IF i_xAlarmReset THEN
	o_xAlarmMotor := FALSE;
END_IF

//sim van janno
//niks

//blinking error van tessa
IF xError THEN
	fbBlinking(io_xBlinking:= o_xErrorMotor);
ELSIF NOT xError AND o_xAlarmMotor THEN
	o_xErrorMotor := TRUE;
ELSE
	o_xErrorMotor := FALSE;
END_IF;

//reset alarm
IF i_xAlarmReset AND NOT xError THEN
	o_xAlarmMotor := FALSE;
END_IF

END_FUNCTION_BLOCK

// ---- POUs/FB_Schuif.TcPOU
FUNCTION_BLOCK FB_Schuif
(*
	Possible options for better code:
	- Errorhandler Method
	- Timer for simulation
*)
VAR_INPUT
	i_eState 				: eSingleState;
	i_eMode					: eModus;
	
	i_xMove					: BOOL; // Start moving to push
	i_xMovePossible			: BOOL; // Is there room on the conveyor? 
	i_xMoveHome				: BOOL; // Move to Home Position
	
	i_xEndSwitchIn			: BOOL;
	i_xEndSwitchOut			: BOOL;
	
	i_xAlarmReset			: BOOL;
	i_xHMIMoveIn: BOOL;
	i_xHMIMoveOut: BOOL;
	i_xHMIStopMoving: BOOL;
END_VAR
VAR_OUTPUT
	o_xMotor 			: BOOL := FALSE;
	o_xMotorDirection	: BOOL;			 // 0 = Going In, 1 = Going Out
	
	o_xErrorSlide 		: BOOL := FALSE; 
	o_xAlarmSlide		: BOOL := FALSE;
	
	o_xMoveDone			: BOOL;
	o_eSlidePosition	: eSlideposition;
END_VAR
VAR
	eSchuifState : eSchuifStates := eSchuifStates.Idle;
	TimerUnknownPos : TON;
	timTimerValue	: TIME := T#20S;
	fbBlikjesBand: FB_BlikjesBand;
END_VAR

// Yvo
TimerUnknownPos(IN := (o_eSlidePosition = eSlideposition.Unknown), PT := timTimerValue);

THIS^.SlidePosition();
THIS^.Simulation();

CASE i_eMode OF
	eModus.Auto :
	CASE i_eState OF
		eSingleState.Execute :
			CASE eSchuifState OF
				eSchuifStates.Idle : // Wait for command
					IF i_xMoveHome THEN
						eSchuifState := eSchuifStates.MovingHome;
					END_IF
					
					IF i_xMove THEN
						eSchuifState := eSchuifStates.MoveOut;
					END_IF
					
				eSchuifStates.MovingHome : // Move Home
					THIS^.MoveHome();
					
				eSchuifStates.MoveOut : // Move out
					THIS^.MoveOut();
					
				eSchuifStates.WaitingForConveyor : // Wait for conveyor
					THIS^.WaitForConveyor();
					
			END_CASE
			
		eSingleState.Suspending :
			// Go to Home
			o_xMotor := TRUE;
			o_xMotorDirection := 0;
			IF i_xEndSwitchIn THEN
				o_xMotor := FALSE;
				o_xMoveDone := FALSE;
			END_IF
			
		eSingleState.Suspended :
			// Go to Home
			o_xMotor := TRUE;
			o_xMotorDirection := 0;
			IF i_xEndSwitchIn THEN
				o_xMotor := FALSE;
				o_xMoveDone := FALSE;
			END_IF
		
		eSingleState.Stopping :
			o_xMotor := TRUE;
			o_xMotorDirection := 0;
			IF i_xEndSwitchIn THEN
				o_xMotor := FALSE;
				o_xMoveDone := FALSE;
			END_IF
			
		eSingleState.Stopped :
			o_xMotor := TRUE;
			o_xMotorDirection := 0;
			IF i_xEndSwitchIn THEN
				o_xMotor := FALSE;
				o_xMoveDone := FALSE;
			END_IF
			
		eSingleState.Aborting :
			o_xMotor := FALSE;
			
		eSingleState.Aborted :
			o_xMotor := FALSE;
			
	END_CASE
	
	eModus.Manual :
		// Doe effe zelf																			// TOEVOEGEN MET HMI
		THIS^.ManualControl();
		
	eModus.Off :
		// Doe niks
		o_xMotor 			:= FALSE;
		
END_CASE

/////////////////
//ERRORHANDLING//
/////////////////
IF TimerUnknownPos.Q THEN
	o_xErrorSlide := TRUE;
	o_xAlarmSlide := TRUE;
END_IF

IF i_xAlarmReset THEN
	o_xErrorSlide := FALSE;
	o_xAlarmSlide := FALSE;
END_IF


// FunctionBlock BlikjesBand
fbBlikjesBand(
	i_xAbort:= , 
	i_eStartStop:= , 
	i_eModus:= , 
	i_xLightSensor:= , 
	i_xAlarmReset:= , 
	i_eNextState:= , 
	i_xManualMotor:= , 
	o_eState=> , 
	o_xMotor=> , 
	o_xWarningFull=> , 
	o_xAcceptingCans=> i_xMovePossible);

METHOD ManualControl : BOOL
VAR_INPUT
END_VAR
IF i_xHMIMoveIn THEN
	THIS^.MoveHome();
ELSIF i_xHMIMoveOut THEN
	o_xMotor := TRUE;
	o_xMotorDirection := 1;
	IF i_xEndSwitchOut THEN
		o_xMotor := FALSE;
		eSchuifState := eSchuifStates.Idle;
	END_IF
ELSIF i_xHMIStopMoving THEN
	o_xMotor := FALSE;
END_IF
END_METHOD

METHOD MoveHome : BOOL
VAR_INPUT
END_VAR
o_xMotor := TRUE;
o_xMotorDirection := 0;
IF i_xEndSwitchIn THEN
	o_xMotor := FALSE;
	o_xMoveDone := FALSE;
	eSchuifState := eSchuifStates.Idle;
END_IF
END_METHOD

METHOD MoveOut : BOOL
VAR_INPUT
END_VAR
IF i_xMovePossible THEN
	o_xMotor := TRUE;
	o_xMotorDirection := 1;
	IF i_xEndSwitchOut THEN
		o_xMoveDone := TRUE;
		eSchuifState := eSchuifStates.MovingHome;
	END_IF
ELSE
	eSchuifState := eSchuifStates.WaitingForConveyor;
END_IF
END_METHOD

METHOD Simulation : BOOL
VAR_INPUT
END_VAR

VAR
	TimerSlideMovement: TON;
	timSlideTimerValue: TIME := T#5S;
END_VAR
//TimerSlideMovement(IN := o_xMotor, PT := timSlideTimerValue);

//IF TimerSlideMovement.Q THEN
	IF o_xMotorDirection = 0 AND o_xMotor THEN
		i_xEndSwitchIn := TRUE;
		i_xEndSwitchOut := FALSE;
	ELSIF o_xMotorDirection = 1 AND o_xMotor THEN
		i_xEndSwitchOut := TRUE;
		i_xEndSwitchIn := FALSE;
	END_IF
//END_IF
END_METHOD

METHOD SlidePosition : BOOL
VAR_INPUT
END_VAR
IF i_xEndSwitchIn AND i_xEndSwitchOut THEN
	o_eSlidePosition := eSlideposition.Unknown;
ELSIF i_xEndSwitchIn THEN
	o_eSlidePosition := eSlideposition.In;
ELSIF i_xEndSwitchOut THEN
	o_eSlidePosition := eSlideposition.Out;
ELSE
	o_eSlidePosition := eSlideposition.Unknown;
END_IF
END_METHOD

METHOD WaitForConveyor : BOOL
VAR_INPUT
END_VAR
o_xMotor := FALSE;
IF i_xMovePossible THEN
	eSchuifState := eSchuifStates.MoveOut;
END_IF
END_METHOD

END_FUNCTION_BLOCK

// ---- POUs/FB_Zuiger.TcPOU
FUNCTION_BLOCK FB_Zuiger
VAR_INPUT
	i_eState 			: eSingleState;
	i_eModes			: eModus := eModus.Auto;
	i_xMoveCiliderDown	: BOOL;
	i_xHallSensorIn		: BOOL;
	i_xHallSensorOut	: BOOL;
	i_xEndSwitchIn		: BOOL;
	i_xEndSwitchOut		: BOOL;
	i_rPressureSensor	: REAL; 
	i_xAlarmResetCilinder	: BOOL;
	i_xAlarmResetAlarmHorizontalMovement	: BOOL;
	i_xAlarmResetPressure : BOOL;
	i_xButtonManStopall : BOOL;
	eManCiliderPosition		: eZuigerCilinderposition;
	eManHorizotalPosition	: eZuigerHorizontaal;
	i_xButtonManVacumOn	: BOOL;
END_VAR
VAR_OUTPUT
	o_xMotor 					: BOOL := FALSE;
	o_xMotorDirectionOut		: BOOL;
	o_xErrorHorizontalMovement 	: BOOL := FALSE;
	o_xAlarmHorizontalMovement	: BOOL;
	o_xMagnetValveCilinder		: BOOL := FALSE;
	o_xMagnetValveVacum	: 			BOOL := FALSE;
	o_xErrorCilinder			: BOOL := FALSE;
	o_xAlarmCilinder			: BOOL;
	o_xErrorPressure			: BOOL := FALSE;
	o_xAlarmPressure			: BOOL;
	o_eCiliderPosition			: eZuigerCilinderposition;
	o_eHorizotalPosition		: eZuigerHorizontaal;
END_VAR
VAR
	eWistedCiliderPosition		: eZuigerCilinderposition;
	eWistedHorizotalPosition	: eZuigerHorizontaal;
	istepcycel : INT;
	TimerCilinder : TON;
	timTimerValue : TIME := T#10S;
	xTimerCilinderRunning: BOOL;
	TimerHorizontal : TON;
	xTimerHorizontalRunning: BOOL;
	
	rPressure_bar: REAL ;
	rMaxbarsensor: REAL := 6;
	rlowpressure: REAL := 4;
	
	
	SIMFUNCTIONING : BOOL := 1;
	o_sStateString: STRING(30);
	xErrorPressure: BOOL;
	xErrorCilinder: BOOL;
	xErrorHorizontalMovement : BOOL;
	fbBlinking : FB_Blinking;
END_VAR

//Timers
TimerCilinder(IN:=xTimerCilinderRunning, PT := timTimerValue);
TimerHorizontal(IN:=xTimerHorizontalRunning, PT := timTimerValue);
CASE i_eModes OF
	eModus.Off:
		StopALL(); //stopall
	eModus.Auto:
		//Case state + control
		CASE i_eState OF
		eSingleState.Aborting:
			StopALL(); //stopall
		eSingleState.Aborted:
			StopALL(); //stopall
		eSingleState.Execute:
			IF i_xMoveCiliderDown=1 AND istepcycel=0 THEN
				istepcycel:=1;
			END_IF
			IF 	o_xAlarmPressure=0 THEN
				CompleetCycel(); //do a compleet cycel
			END_IF
		eSingleState.Idle:
			istepcycel:=0;
			CiliderUP(); //to startingpostion
			IF o_eCiliderPosition = eZuigerCilinderposition.Up THEN
				HorizontalIN();
			END_IF
		eSingleState.Stopping:
			istepcycel:=0;
			CiliderUP(); //to startingpostion
			IF o_eCiliderPosition = eZuigerCilinderposition.Up THEN
				HorizontalIN();
			END_IF
		eSingleState.Stopped:
			istepcycel:=0;
			CiliderUP(); //to startingpostion
			IF o_eCiliderPosition = eZuigerCilinderposition.Up THEN
				HorizontalIN();
			END_IF
		eSingleState.Suspending:
			istepcycel:=0;
			CiliderUP(); //to startingpostion
			IF o_eCiliderPosition = eZuigerCilinderposition.Up THEN
				HorizontalIN();
			END_IF
		eSingleState.Suspended:
			istepcycel:=0;
			CiliderUP(); //to startingpostion
			IF o_eCiliderPosition = eZuigerCilinderposition.Up THEN
				HorizontalIN();
			END_IF
		END_CASE
	eModus.Manual: //manual controll
		IF i_xButtonManStopall THEN
			StopALL(); //stopall
		ELSIF eManCiliderPosition =  eZuigerCilinderposition.up THEN
			CiliderUP(); //to startingpostion
		ELSIF eManCiliderPosition =  eZuigerCilinderposition.Down THEN
			CilinderDOwn();
		END_IF
		IF NOT i_xButtonManStopall AND eManHorizotalPosition	= eZuigerHorizontaal.In THEN
			HorizontalIN();
		ELSIF NOT i_xButtonManStopall AND eManHorizotalPosition	= eZuigerHorizontaal.Out THEN
			HoriztalOUT();
		END_IF
		IF NOT i_xButtonManStopall AND NOT i_xButtonManVacumOn THEN
			o_xMagnetValveVacum:=FALSE;
		ELSIF NOT i_xButtonManStopall AND i_xButtonManVacumOn THEN
			o_xMagnetValveVacum:=TRUE;
		END_IF
END_CASE

//Errors
IF  NOT (eWistedCiliderPosition = o_eCiliderPosition) THEN //error timer cilinder
	xTimerCilinderRunning:=1;
ELSE
	xTimerCilinderRunning:=0;
END_IF

IF TimerCilinder.Q THEN //error cilinder when timer gone
	xErrorCilinder:=1;
	o_xAlarmCilinder:=1;
ELSE
	xErrorCilinder:=0;
END_IF

IF xErrorCilinder THEN
	fbBlinking(io_xBlinking:= o_xErrorCilinder);
ELSIF NOT xErrorCilinder AND o_xAlarmCilinder THEN
	o_xErrorCilinder := TRUE;
ELSE
	o_xErrorCilinder := FALSE;
END_IF;


IF  (NOT (eWistedHorizotalPosition = o_eHorizotalPosition)) AND o_xMotor THEN //error start timer horizonal
	xTimerHorizontalRunning:=1;
ELSE
	xTimerHorizontalRunning:=0;
END_IF

IF TimerHorizontal.Q THEN
	xErrorHorizontalMovement:=1;
	o_xAlarmHorizontalMovement:=1;
ELSE
	xErrorHorizontalMovement:=0;
END_IF

IF xErrorHorizontalMovement THEN
	fbBlinking(io_xBlinking:= o_xErrorHorizontalMovement);
ELSIF NOT xErrorHorizontalMovement AND o_xAlarmHorizontalMovement THEN
	o_xErrorHorizontalMovement := TRUE;
ELSE
	o_xErrorHorizontalMovement := FALSE;
END_IF;

//pressuresensor error
rPressure_bar := (i_rPressureSensor / 4095.0) * rMaxbarsensor;// 4095 form analog and 6 from 6 bar max from the sensor
IF rPressure_bar<rlowpressure THEN
	xErrorPressure:=1;
	o_xAlarmPressure:=1;
ELSE
	xErrorPressure:=0;
END_IF

IF xErrorPressure THEN
	fbBlinking(io_xBlinking:= o_xErrorPressure);
ELSIF NOT xErrorPressure AND o_xAlarmPressure THEN
	o_xErrorPressure := TRUE;
ELSE
	o_xErrorPressure := FALSE;
END_IF;

//Alarm reset
IF i_xAlarmResetCilinder AND NOT  xErrorCilinder THEN
	o_xAlarmCilinder:=0;
END_IF 
IF NOT 	xErrorHorizontalMovement AND i_xAlarmResetAlarmHorizontalMovement THEN
	o_xAlarmHorizontalMovement:=0;
END_IF
IF NOT xErrorPressure AND  i_xAlarmResetPressure THEN
	o_xAlarmPressure:=0;
END_IF

//actualpostioncilinder
IF	i_xHallSensorIn AND i_xHallSensorOut THEN
	o_eCiliderPosition := eZuigerCilinderposition.Unkown;
ELSIF i_xHallSensorIn	THEN
	o_eCiliderPosition := eZuigerCilinderposition.Up;
ELSIF i_xHallSensorOut THEN
	o_eCiliderPosition := eZuigerCilinderposition.Down;
ELSE
	o_eCiliderPosition := eZuigerCilinderposition.Unkown;
END_IF

//actualpostionhorizontal with motor controll
IF	i_xEndSwitchIn AND i_xEndSwitchOut THEN
	o_eHorizotalPosition := eZuigerHorizontaal.Unkown;
ELSIF i_xEndSwitchIn	THEN
	o_eHorizotalPosition := eZuigerHorizontaal.In;
ELSIF i_xEndSwitchOut THEN
	o_eHorizotalPosition := eZuigerHorizontaal.Out;
ELSE
	o_eHorizotalPosition := eZuigerHorizontaal.Unkown;
END_IF

IF eWistedHorizotalPosition = o_eHorizotalPosition THEN
	o_xMotor:=0;
ELSIF NOT (eWistedHorizotalPosition = o_eHorizotalPosition) THEN
	o_xMotor:=1;
END_IF

SIM();
o_sStateString := F_StateEnumToStringSingleState(i_eState);

METHOD PRIVATE CiliderUP
//moves the cilider up
eWistedCiliderPosition :=eZuigerCilinderposition.Up;
o_xMagnetValveCilinder:=0;
END_METHOD

METHOD PRIVATE CilinderDOwn
VAR_INPUT
END_VAR
//moves the cilider Down
eWistedCiliderPosition :=eZuigerCilinderposition.Down;
o_xMagnetValveCilinder:=1;
END_METHOD

METHOD PRIVATE CompleetCycel
VAR

END_VAR
	o_eHorizotalPosition := eZuigerHorizontaal.In;
		o_eCiliderPosition := eZuigerCilinderposition.Unkown;
		

CASE istepcycel OF
	1: //too startingpostition
		o_xMagnetValveVacum:=FALSE;
		CiliderUP();
		IF o_eCiliderPosition = eZuigerCilinderposition.Up THEN
			HorizontalIN();
		END_IF
		IF o_eCiliderPosition = eZuigerCilinderposition.Up AND o_eHorizotalPosition =eZuigerHorizontaal.IN THEN
			istepcycel:=2;
		END_IF
	2: 		//zuiger naar beneden totdat beneden
		o_xMagnetValveVacum:=TRUE;
		CilinderDOwn();
		IF o_eCiliderPosition = eZuigerCilinderposition.DOWN THEN
			istepcycel:=3;
		END_IF
	3: //zuiger omhoog
		o_xMagnetValveVacum:=TRUE;
		CiliderUP();
		IF o_eCiliderPosition = eZuigerCilinderposition.UP THEN
			istepcycel:=4;
		END_IF
	4:
		o_xMagnetValveVacum:=TRUE;
		HoriztalOUT();
		IF o_eHorizotalPosition = eZuigerHorizontaal.OUT THEN
				istepcycel:=5;
		END_IF
	5:	
		o_xMagnetValveVacum:=FALSE;
		HorizontalIN();
		IF o_eHorizotalPosition = eZuigerHorizontaal.IN THEN
				istepcycel:=0;
		END_IF

END_CASE
END_METHOD

METHOD PRIVATE HorizontalIN
VAR_INPUT
END_VAR

o_xMotorDirectionOut:=0;
eWistedHorizotalPosition := eZuigerHorizontaal.In;
END_METHOD

METHOD PRIVATE HoriztalOUT
VAR_INPUT
END_VAR
//hoizontal out


o_xMotorDirectionOut:=1;
eWistedHorizotalPosition := eZuigerHorizontaal.Out;
END_METHOD

METHOD SIM
VAR

END_VAR
//simulatie
IF gvl.g_xSimulationActive THEN
	IF SIMFUNCTIONING THEN
		

		IF GVL.TimerShort.Q THEN
			i_rPressureSensor := 4000;
			IF o_xMagnetValveCilinder THEN //simulation
				i_xHallSensorIn := FALSE;
				i_xHallSensorOut := TRUE;
			ELSIF NOT o_xMagnetValveCilinder THEN
				i_xHallSensorIn := TRUE;
				i_xHallSensorOut := FALSE;
			END_IF
		END_IF
		
		IF GVL.Timerlong.Q THEN		
			IF o_xMotor AND o_xMotorDirectionOut THEN
				i_xEndSwitchIn := FALSE;
				i_xEndSwitchOut := TRUE;
			ELSIF o_xMotor AND NOT o_xMotorDirectionOut THEN
				i_xEndSwitchIn := TRUE;
				i_xEndSwitchOut := FALSE;
			END_IF
		END_IF
		
	END_IF
	
END_IF
END_METHOD

METHOD PRIVATE StopALL : BOOL
VAR_INPUT
END_VAR
o_xMagnetValveCilinder:=0;
eWistedHorizotalPosition := o_eHorizotalPosition;

IF	i_xHallSensorIn AND i_xHallSensorOut THEN
	o_eCiliderPosition := eZuigerCilinderposition.Unkown;
ELSIF i_xHallSensorIn	THEN
	o_eCiliderPosition := eZuigerCilinderposition.Up;
ELSIF i_xHallSensorOut THEN
	o_eCiliderPosition := eZuigerCilinderposition.Down;
ELSE
	o_eCiliderPosition := eZuigerCilinderposition.Unkown;
END_IF
//i want to dont like this
//eWistedHorizotalPosition = o_eHorizotalPosition;

IF	i_xEndSwitchIn AND i_xEndSwitchOut THEN
	o_eHorizotalPosition := eZuigerHorizontaal.Unkown;
ELSIF i_xEndSwitchIn	THEN
	o_eHorizotalPosition := eZuigerHorizontaal.In;
ELSIF i_xEndSwitchOut THEN
	o_eHorizotalPosition := eZuigerHorizontaal.Out;
ELSE
	o_eHorizotalPosition := eZuigerHorizontaal.Unkown;
END_IF
END_METHOD

END_FUNCTION_BLOCK

// ---- POUs/FB_LiftA_Extended.TcPOU
FUNCTION_BLOCK FB_LiftA_Extended EXTENDS FB_Lift

VAR_INPUT
	i_aLayerHeights	: ARRAY[1..10] OF INT;
	i_iLayerCount: INT;
	i_eZuigerDone : eZuigerCilinderPosition;
END_VAR

VAR_OUTPUT
	o_xGoSchuif: BOOL;
	o_xGoZuiger: BOOL;
END_VAR

VAR
	LayerState: INT;
	LiftASteps:	INT;
END_VAR

SUPER^();
iConveyorHeight := iHomePosition;

CASE i_eMode OF
	eModus.Auto :
	//////////////////////////////////////////////////////////////////////////
		CASE i_eState OF
			eSingleState.Execute :
				IF i_xPalletInPosition THEN
					CASE LiftASteps OF
						1:
							THIS^.Impale();
							IF o_ePinsPositions = eLiftPins.Out THEN
								LiftASteps := 2;
							END_IF
						2:
							IF i_xMoveUpSafe THEN
								LiftASteps := 3;
							END_IF
						3:
							THIS^.MoveUpToLayer();
					END_CASE
				END_IF
		END_CASE
	//////////////////////////////////////////////////////////////////////////
	eModus.Manual :
		// Doe effe zelf																			// TOEVOEGEN MET HMI
		// Lift handmatig bedienen door INT invoer?
		// Pins handmatig in en uit, met beveiliging zodat pallet niet naar beneden dondert
	eModus.Off :
		// Doe niks
		// Stop
		o_xMotor := FALSE;
END_CASE

METHOD MoveHome : BOOL
VAR_INPUT
END_VAR
CASE InitHomeStates OF
	0 :	// Start Homing if the endswitch isnt active.
		IF NOT i_xEndSwitch THEN
        	InitHomeStates := 1;
		ELSE 
			// Already at home position
			o_xMotor := FALSE;
			InitHomeStates := 4;
    	END_IF
	
	1 :	// Go to conveyorheight
		o_xMotor := TRUE;
		o_iTargetPos := iHomePosition;
		
		IF i_iServoEncoder = o_iTargetPos THEN
			o_xMotor := FALSE;                  // stop motion
			InitHomeStates := 2;
		END_IF
		
	2 : 
		// Home
END_CASE
END_METHOD

METHOD MoveUpToLayer : BOOL
VAR_INPUT
END_VAR

VAR
	CurrentLayer: INT;
END_VAR
CASE LayerState OF
	0: // Idle / Start
		o_xLiftDone := FALSE;
		CurrentLayer := 1;
	
		IF i_iLayerCount > 0 THEN
			LayerState := 1;
		END_IF
	
	
	1: // Move to current layer
		o_iTargetPos := i_aLayerHeights[CurrentLayer];
		o_xMotor := TRUE;
	
		IF i_iServoEncoder = o_iTargetPos THEN
			o_xMotor := FALSE;
			LayerState := 2;
		END_IF
	
	
	2: // Do action at layer
		o_xGoZuiger := TRUE;	// Use Zuiger to remove any layer cartons
		IF i_eZuigerDone = eZuigerCilinderPosition.Up THEN
			o_xGoSchuif := TRUE;	// Push cans onto conveyor
		END_IF
		
		IF i_xMoveUpSafe THEN
			o_xGoZuiger := FALSE;
			o_xGoSchuif := FALSE;
			LayerState := 3;
		END_IF
	
	3: // Advance to next layer
		CurrentLayer := CurrentLayer + 1;
	
		IF CurrentLayer > i_iLayerCount THEN
			LayerState := 4;   // all layers done
		ELSE
			LayerState := 1;   // go to next layer
		END_IF
	
	
	4: // Finished
		o_xLiftDone := TRUE;
		THIS^.MoveHome();
		// wait here

END_CASE
END_METHOD

END_FUNCTION_BLOCK

// ---- POUs/FB_Lift.TcPOU
FUNCTION_BLOCK FB_Lift
VAR_INPUT
	i_eState 			: eSingleState;
	i_eMode				: eModus := eModus.Auto;
	i_eLiftState		: eLiftStates;
	
	i_iServoEncoder 	: INT;
	
	i_xEndSwitch		: BOOL;
	
	i_xPin1HallSensorIn	: BOOL;
	i_xPin2HallSensorIn	: BOOL;
	i_xPin3HallSensorIn	: BOOL;
	i_xPin4HallSensorIn	: BOOL;
	
	i_xPin1HallSensorOut	: BOOL;
	i_xPin2HallSensorOut	: BOOL;
	i_xPin3HallSensorOut	: BOOL;
	i_xPin4HallSensorOut	: BOOL;
	
	i_xLightSensor1 : BOOL;
	i_xLightSensor2 : BOOL;
	
	i_xMoveUpSafe: BOOL;
	i_xMoveDownSafe: BOOL;
	i_xPalletInPosition: BOOL;
END_VAR
VAR_OUTPUT
	o_iTargetPos		: INT;
	o_eLiftPosition		: ELIFTPOSITION;
	o_xMotor			: BOOL;
	o_xMagnetValve		: BOOL;
	o_ePinsPositions	: eLiftPins;
	o_xLiftDone			: BOOL;
END_VAR
VAR
	iConveyorHeight: INT;
	iHomePosition: INT;
	iImpaleErrorCounter: INT;
	InitHomeStates: INT;
END_VAR

THIS^.CheckPins();
THIS^.LiftPosition();
THIS^.Simulation();
THIS^.ErrorHandler();


CASE i_eLiftState OF
	eLiftStates.InitHome :
		// Initialise Home
		THIS^.InitHome();
	
	eLiftStates.Impale :
		// Impale op de manier van welke lift het is
		THIS^.Impale();

END_CASE

METHOD CheckPins : BOOL
VAR_INPUT
END_VAR
IF i_xPin1HallSensorIn
AND i_xPin2HallSensorIn
AND i_xPin3HallSensorIn
AND i_xPin4HallSensorIn THEN
	o_ePinsPositions := eLiftPins.In;

ELSIF i_xPin1HallSensorOut
AND i_xPin2HallSensorOut
AND i_xPin3HallSensorOut
AND i_xPin4HallSensorOut THEN
	o_ePinsPositions := eLiftPins.Out;
	
ELSE
	o_ePinsPositions := eLiftPins.Unknown;
END_IF
END_METHOD

METHOD ErrorHandler : BOOL
VAR_INPUT
END_VAR

(*
	When can an error occur?
	- Pins are unknown for too long
	- Pins are in or Unknown while pallet is lifted.
*)
// If pins are in or unknown while pallet is lifted, fatal error.
IF i_iServoEncoder > iConveyorHeight AND
	(o_ePinsPositions = eLiftPins.In OR o_ePinsPositions = eLiftPins.Unknown) THEN
	// ERROR PINS
END_IF;
END_METHOD

METHOD Impale : BOOL
VAR_INPUT
END_VAR
o_xMagnetValve := TRUE;

THIS^.CheckPins();

IF o_ePinsPositions = eLiftPins.In OR o_ePinsPositions = eLiftPins.Unknown THEN
	iImpaleErrorCounter := iImpaleErrorCounter + 1;
END_IF
END_METHOD

METHOD InitHome : BOOL
VAR_INPUT
END_VAR

VAR
END_VAR
CASE InitHomeStates OF
	0 :	// Start Homing if the endswitch isnt active.
		IF NOT i_xEndSwitch THEN
        	InitHomeStates := 1;
		ELSE 
			// Already at home position
			o_xMotor := FALSE;
			iHomePosition := i_iServoEncoder;
			InitHomeStates := 4;
    	END_IF
	
	1 :	// Go to conveyorheight
		o_xMotor := TRUE;
		o_iTargetPos := iConveyorHeight;
		
		IF i_iServoEncoder = o_iTargetPos THEN
			o_xMotor := FALSE;                  // stop motion
			InitHomeStates := 2;
		END_IF
		
	2 : // Release Pallet
		o_xMagnetValve := FALSE;
		
		IF o_ePinsPositions = eLiftPins.In THEN
        	InitHomeStates := 3;
    	END_IF
	
	3 :	// Go down until the endswitch is reached.
		o_xMotor := TRUE;
		o_eLiftPosition := eLiftPosition.GoingDown;
		
		IF i_xEndSwitch THEN
			o_xMotor := FALSE;
			iHomePosition := i_iServoEncoder;
			InitHomeStates := 4;
		END_IF
	
	4 :
		// Home Done
END_CASE
END_METHOD

METHOD LiftPosition : BOOL
VAR_INPUT
END_VAR
IF i_iServoEncoder = o_iTargetPos THEN
	// Idle
	o_eLiftPosition := eLiftPosition.Idle;
ELSIF i_iServoEncoder < o_iTargetPos THEN
	// Going Up
	o_eLiftPosition := eLiftPosition.GoingUp;
ELSIF i_iServoEncoder > o_iTargetPos THEN
	// Going Down
	o_eLiftPosition := eLiftPosition.GoingDown;
ELSIF i_xEndSwitch THEN
	o_eLiftPosition := eLiftPosition.Home;
END_IF
END_METHOD

METHOD Simulation : BOOL
VAR_INPUT
END_VAR
IF o_eLiftPosition = eLiftPosition.GoingUp AND o_xMotor = TRUE THEN
	i_iServoEncoder := i_iServoEncoder + 1;
ELSIF o_eLiftPosition = eLiftPosition.GoingDown AND o_xMotor = TRUE THEN
	i_iServoEncoder := i_iServoEncoder - 1;
END_IF
END_METHOD

END_FUNCTION_BLOCK

// ---- POUs/FB_Palletizer.TcPOU
FUNCTION_BLOCK FB_Palletizer
VAR_INPUT
	i_xAbort		 	: BOOL;
	i_eStartStop 		: eStartStop;
	i_PreviousEmptying	: BOOL;
	i_xDoorOpenButton	: BOOL;	
	i_xWarningReset		: BOOL;
	i_eModus			: eModus := eModus.Auto;
	i_xPalletsEmptyed: BOOL;
END_VAR
VAR_OUTPUT
	o_eState 			: eSingleState;
	o_iStorageCount		: INT;
	o_xWarningFull		: BOOL;
	o_xExpectingPallet	: BOOL;
END_VAR
VAR
	
	fbBand	: FB_Band;
	TimerLift: TON;
	xTimerLiftRunning: BOOL;
	timTimerValue: TIME :=T#10S;
	xGoHoldBand : BOOL;
	xGoEmptyBand : BOOL;
	istep		: INT;
	ximpaled : BOOL;
	fbLiftB: FB_LiftB_Extended;
	xAuto : BOOL;
	TimerAcceptingPallet : ton;
	xTimerEmtyingRunning: BOOL;
	timTimerValueemtying: TIME;
	o_sStateString: STRING(30);
	xpreviuosEmtyed: BOOL;
	xPalletIn: BOOL;
	
	rMotorOff: F_TRIG;
END_VAR

//timer for error
TimerAcceptingPallet(IN:=xpreviuosEmtyed, PT := timTimerValue);

rMotorOff(CLK := fbLiftB.o_xMotor);


//calling band and giving corect stuf
fbBand(
	i_eState:= o_eState, 
	i_xGoHold:= xGoHoldBand, 
	i_xGoEmpty:= xGoEmptyBand, 
	i_xAlarmReset:= , 
	o_xMotor=> , 
	o_xErrorMotor=> , 
	o_xAlarmMotor=> , 
	o_xGivingToNext=> );

fbLiftB(
	i_eState:= o_eState, 
	i_eMode:= , 
	i_eLiftState:= , 
	i_iServoEncoder:= , 
	i_xEndSwitch:= , 
	i_xPin1HallSensorIn:= , 
	i_xPin2HallSensorIn:= , 
	i_xPin3HallSensorIn:= , 
	i_xPin4HallSensorIn:= , 
	i_xPin1HallSensorOut:= , 
	i_xPin2HallSensorOut:= , 
	i_xPin3HallSensorOut:= , 
	i_xPin4HallSensorOut:= , 
	i_xLightSensor1:= , 
	i_xLightSensor2:= , 
	i_xMoveUpSafe:= , 
	i_xMoveDownSafe:= , 
	i_xPalletInPosition:= , 
	o_iTargetPos=> , 
	o_eLiftPosition=> , 
	o_xMotor=> , 
	o_xMagnetValve=> , 
	o_ePinsPositions=> , 
	o_xLiftDone=> , 
	i_iMoveToLayer:= );
	

fbLiftB();
fbLiftB.i_eState:=o_eState;
//calling lift

IF	fbLiftB.i_xPin1HallSensorIn AND NOT //when inpaled and when not
	fbLiftB.i_xPin1HallSensorOut AND
	fbLiftB.i_xPin2HallSensorIn AND NOT
	fbLiftB.i_xPin2HallSensorOut AND
	fbLiftB.i_xPin3HallSensorIn AND NOT
	fbLiftB.i_xPin3HallSensorOut AND
	fbLiftB.i_xPin4HallSensorIn AND NOT
	fbLiftB.i_xPin4HallSensorOut AND 
	ximpaled THEN
	ximpaled:=0;
ELSIF NOT fbLiftB.i_xPin1HallSensorIn AND 
	fbLiftB.i_xPin1HallSensorOut AND NOT
	fbLiftB.i_xPin2HallSensorIn AND 
	fbLiftB.i_xPin2HallSensorOut AND NOT
	fbLiftB.i_xPin3HallSensorIn AND 
	fbLiftB.i_xPin3HallSensorOut AND NOT
	fbLiftB.i_xPin4HallSensorIn AND 
	fbLiftB.i_xPin4HallSensorOut AND NOT
	ximpaled THEN
	ximpaled:=1;
END_IF

IF i_eModus<2 THEN//when to abort
	IF  o_eState<7 AND (i_xAbort OR fbBand.o_xErrorMotor OR fbLiftB.o_xErrorLift OR fbLiftB.o_xErrorImpaler) THEN 
		o_eState := eSingleState.Aborting;
	ELSIF o_eState = eSingleState.Execute AND (o_xWarningFull OR i_xDoorOpenButton)  THEN //when to suspend
		o_eState := eSingleState.Suspending;
	END_IF
END_IF
//state code
CASE o_eState OF
	eSingleState.Idle://start
		
			o_eState := eSingleState.Execute;
		
	
	eSingleState.Execute:
		// Door opened -> suspend machine
		// Stop button pressed
		IF i_eStartStop = eStartStop.Stop  AND o_eState = eSingleState.Execute THEN
			o_eState := eSingleState.Stopping;
		END_IF
		IF xAuto THEN //if auto function auto
			CASE istep OF
						0:
						//start position
							xGoHoldBand := TRUE;
							xGoEmptyBand := FALSE;//stop band
							o_xExpectingPallet := 0;//not expecting
							//lift in start
							fbLiftB.i_iMoveToLayer:=1;
							IF NOT fbBand.o_xMotor AND NOT fbLiftB.o_xMotor THEN //if band and lift stopted
								fbLiftB.i_eLiftState:= eLiftStates.Deimpale;
								istep:=1;
							END_IF
						1:
						//accepting pallet
							IF NOT xPalletIn THEN
								o_xExpectingPallet := 1;
								IF i_PreviousEmptying AND NOT TimerAcceptingPallet.q THEN //start band if pervious emtying
									xGoHoldBand := FALSE;
									xGoEmptyBand := TRUE;
									xpreviuosEmtyed:=1; 
								ELSIF TimerAcceptingPallet.q THEN
									istep:=2;
									xGoHoldBand := TRUE;
									xGoEmptyBand := FALSE;
									o_xExpectingPallet:=0;
									xpreviuosEmtyed:=0;
								END_IF
							ELSE
								
								istep:=2;
							END_IF
								
							
						2:
						//position witch pallet
						
							
								//from position to impaling
								IF NOT ximpaled AND (fbLiftB.i_iMoveToLayer>1 OR fbLiftB.i_iMoveToLayer=0) THEN // if not holding pallet and not in postion to impale
									
									fbLiftB.i_iMoveToLayer:=1;

	
								ELSIF NOT ximpaled AND (fbLiftB.i_iMoveToLayer=1) THEN //if the impaler is not holding a pallet and ther is a nieuw pallet and its in position  to pik it up
									IF  NOT fbLiftB.o_xMotor THEN//and lift
										fbLiftB.i_eLiftState:= eLiftStates.Impale;
										o_xExpectingPallet:=0;
										
										istep:=3;
									END_IF
								end_if
	
								IF  ximpaled AND (fbLiftB.i_iMoveToLayer>1) THEN //if holding pallet and there is a nieuw pallet
									fbLiftB.i_iMoveToLayer:=3;
									IF rMotorOff.Q AND fbLiftB.i_iMoveToLayer=3 THEN//and lift
										fbLiftB.i_eLiftState:= eLiftStates.Deimpale;//moet deimpale zijn maar bestaat niet
									END_IF
								END_IF
	
						
						3:
						//holding and accepting pallets
						IF ximpaled THEN //is holding pallet
							xGoHoldBand := TRUE;
							xGoEmptyBand := FALSE;
							fbLiftB.i_iMoveToLayer:=2;
							//move to holding
							IF rMotorOff.Q AND fbLiftB.i_iMoveToLayer=2 THEN
								
								IF xPalletIn=0 THEN
								o_iStorageCount:=o_iStorageCount+1;
								END_IF
								xPalletIn:=0;
								istep:=1;
							END_IF
						END_IF
				END_CASE
			END_IF
		//normal opperation
		CASE i_eModus OF
			eModus.Auto:
				xAuto:=1;
				//
			eModus.Manual:
				xAuto:=0;
				istep:=0;
			eModus.Off:
			IF istep=1 THEN
				xAuto:=0;
				IF o_eState=eSingleState.Execute THEN
					o_eState := eSingleState.Stopping;
				END_IF
			END_IF

		END_CASE
		
		
		

	eSingleState.Stopping: //
		// Stop band movement
		o_xExpectingPallet:=0;
		xGoHoldBand := TRUE;
		xGoEmptyBand := FALSE;
		IF fbLiftB.i_iMoveToLayer>1 THEN
			fbLiftB.i_iMoveToLayer:=1;
			IF  rMotorOff.Q AND fbLiftB.i_iMoveToLayer=1 THEN//and lift
				fbLiftB.i_eLiftState:= eLiftStates.Deimpale;//has to be deinmpale but does not yet eqzist
			END_IF
		END_IF
		
		IF NOT ximpaled AND (fbLiftB.i_iMoveToLayer=1 OR fbLiftB.i_iMoveToLayer=0) THEN
			fbLiftB.i_iMoveToLayer:=0;
			IF  NOT fbLiftB.o_xMotor AND fbLiftB.i_iMoveToLayer=0 THEN//and lift
				IF o_iStorageCount>0 THEN
					xPalletIn:=1;
				END_IF
				istep:=0;
				o_eState := eSingleState.Stopped;
				
			END_IF
		END_IF

		IF i_xAbort THEN
			o_eState := eSingleState.Aborting;
		END_IF

	eSingleState.Stopped:
		// All movements stopped
		o_xExpectingPallet:=0;
		IF xAuto AND i_eStartStop = eStartStop.Start THEN
			o_eState := eSingleState.Execute;
		END_IF

		IF i_xAbort THEN
			o_eState := eSingleState.Aborting;
		END_IF

	eSingleState.Suspending:
		o_xExpectingPallet:=0;
		// Stop band movement
		xGoHoldBand := TRUE;
		xGoEmptyBand := FALSE;
		IF  ximpaled AND ( NOT (fbLiftB.i_iMoveToLayer=0) OR NOT (fbLiftB.i_iMoveToLayer=1)) THEN
			fbLiftB.i_iMoveToLayer:=1;
			IF  rMotorOff.Q AND fbLiftB.i_iMoveToLayer=1 THEN//and lift
				fbLiftB.i_eLiftState:= eLiftStates.Deimpale;//moet deimpale zijn maar bestaat niet
			END_IF
		ELSIF ximpaled AND  (fbLiftB.i_iMoveToLayer=1) THEN
			fbLiftB.i_eLiftState:= eLiftStates.Deimpale;
		END_IF
		
		IF NOT ximpaled THEN
			fbLiftB.i_iMoveToLayer:=0;
			IF  NOT fbLiftB.o_xMotor AND fbLiftB.i_iMoveToLayer=0 THEN//and lift
				istep:=0;
				o_eState := eSingleState.Suspended;
			END_IF
		END_IF


		IF i_xAbort THEN
			o_eState := eSingleState.Aborting;
		END_IF



	eSingleState.Suspended:
		// Machine is safe, waiting
		o_xExpectingPallet:=0;
		IF i_xPalletsEmptyed THEN
			o_iStorageCount:=0;
		END_IF
		IF NOT i_xDoorOpenButton THEN
			//xTimerEmtyingRunning:=1;
			IF o_iStorageCount<8 AND NOT o_xWarningFull THEN
				IF o_iStorageCount>0 THEN
					xPalletIn:=1;
				END_IF
				istep := 0;
				o_eState := eSingleState.Execute;
				//xTimerEmtyingRunning:=0;
			END_IF

		END_IF





	eSingleState.Aborting:
		o_xExpectingPallet:=0;
		// Immediately stop band
		xGoHoldBand := TRUE;
		xGoEmptyBand := FALSE;

		// Lift: immediately stop movement
		// Lift stops immediately at current position

		// When everything is stopped
		IF NOT fbBand.o_xMotor AND NOT fbLiftB.o_xMotor THEN
			o_eState := eSingleState.Aborted;
		END_IF



	eSingleState.Aborted:
		o_xExpectingPallet:=0;
		// Machine is halted due to abort or alarm

		IF NOT i_xAbort AND NOT o_xWarningFull AND NOT fbBand.o_xErrorMotor AND NOT fbLiftB.o_xErrorLift AND NOT fbLiftB.o_xErrorImpaler THEN
			// Reset abort condition
			o_eState := eSingleState.Stopped;
		END_IF


END_CASE
//errors

//allarmen
IF o_iStorageCount = 8 THEN
	o_xWarningFull:=TRUE;
ELSIF i_xWarningReset THEN
	o_xWarningFull:=FALSE;
	o_iStorageCount:=0;
END_IF

//warnings

o_sStateString := F_StateEnumToStringSingleState(o_eState);

//sim sensor lift location
IF i_eModus = eModus.auto OR i_eModus = eModus.Off THEN	
	IF ximpaled THEN
		fbLiftB.i_xLightSensor2:=FALSE;
		fbLiftB.i_xLightSensor2:=TRUE;
	ELSIF i_PreviousEmptying AND istep=1  THEN
		fbLiftB.i_xLightSensor2:=TRUE;
		fbLiftB.i_xLightSensor2:=FALSE;
	ELSIF istep=2 THEN
		fbLiftB.i_xLightSensor2:=FALSE;
		fbLiftB.i_xLightSensor2:=TRUE;
	END_IF
END_IF
//
//help

END_FUNCTION_BLOCK

// ---- POUs/FB_LiftB_Extended.TcPOU
FUNCTION_BLOCK FB_LiftB_Extended EXTENDS FB_Lift
VAR_INPUT
	i_iMoveToLayer : INT;
END_VAR

VAR_OUTPUT
	
END_VAR

VAR
	iPalletizeHeight: INT := iHomePosition + 2000;
	iHighestHeight	: INT := iHomePosition + 3000;
END_VAR

// Janno geeft door naar welke laag hij moet. Laag 0 = home, laag 1 = band, laag 2 = pallet op pallet, laag 3 = pallets hoog

SUPER^(); // Call parent Functionblock
iConveyorHeight := iHomePosition + 1000;

// CASE i_eMode OF
// 	eModus.Auto :
// 	CASE i_eState OF
// 		eSingleState.Execute :
			CASE i_eLiftState OF		
				eLiftStates.MoveUpToLayer :														// Testen
				 	// Ga naar de positie van de volgende laag.
					CASE i_iMoveToLayer OF
						0 :
							// Ga naar home
							THIS^.MoveHome(); 													// Testen
						1 :
							// Ga naar band hoogte
							THIS^.GoToConveyorHeight(); 										// Testen
						2 : 
							// Ga naar stapelhoogte
							THIS^.GoToHighestHeight(); 											// Testen
						3 :
							// Ga hoog
							THIS^.GoToPalletizeHeight(); 										// Testen
					END_CASE
					
				
			END_CASE
// 	END_CASE
	
// 	eModus.Manual :
// 		// Doe effe zelf																			// TOEVOEGEN MET HMI
// 		// Lift handmatig bedienen door INT invoer?
// 		// Pins handmatig in en uit, met beveiliging zodat pallet niet naar beneden dondert
// 	eModus.Off :
// 		// Doe niks
// 		// Stop
// END_CASE

METHOD GoToConveyorHeight : BOOL
VAR_INPUT
END_VAR
o_xMotor := TRUE;
o_iTargetPos := iConveyorHeight;

IF i_iServoEncoder = iConveyorHeight THEN
	o_xMotor := FALSE;
END_IF;
END_METHOD

METHOD GoToHighestHeight : BOOL
VAR_INPUT
END_VAR
o_xMotor := TRUE;
o_iTargetPos := iHighestHeight;

IF i_iServoEncoder = iHighestHeight THEN
	o_xMotor := FALSE;
END_IF;
END_METHOD

METHOD GoToPalletizeHeight : BOOL
VAR_INPUT
END_VAR
o_xMotor := TRUE;
o_iTargetPos := iPalletizeHeight;

IF i_iServoEncoder = iPalletizeHeight THEN
	o_xMotor := FALSE;
END_IF;
END_METHOD

METHOD MoveHome : BOOL
VAR_INPUT
END_VAR
CASE InitHomeStates OF
	0 :	// Start Homing if the endswitch isnt active.
		IF NOT i_xEndSwitch THEN
        	InitHomeStates := 1;
		ELSE 
			// Already at home position
			o_xMotor := FALSE;
			InitHomeStates := 4;
    	END_IF
	
	1 :	// Go to conveyorheight
		o_xMotor := TRUE;
		o_iTargetPos := iConveyorHeight;
		
		IF i_iServoEncoder = o_iTargetPos THEN
			o_xMotor := FALSE;                  // stop motion
			InitHomeStates := 2;
		END_IF
		
	2 : // Release Pallet
		o_xMagnetValve := FALSE;
		
		IF o_ePinsPositions = eLiftPins.In THEN
        	InitHomeStates := 3;
    	END_IF
	
	3 :	// Go down until the endswitch is reached.
		o_xMotor := TRUE;
		o_eLiftPosition := eLiftPosition.GoingDown;
		
		IF i_xEndSwitch THEN
			o_xMotor := FALSE;
			InitHomeStates := 4;
		END_IF
	
	4 :
		// Home Done
END_CASE
END_METHOD

METHOD WaitForPallet : BOOL
VAR_INPUT
END_VAR
// Wait for pallet
END_METHOD

END_FUNCTION_BLOCK

// ---- POUs/FB_LiftJanno.TcPOU
FUNCTION_BLOCK FB_LiftJanno
VAR_INPUT
	i_iMoveToLayer : INT;
	i_eState 			: eSingleState;
	i_eMode				: eModus;
	i_eLiftState 		: eLiftStates;
	
	i_xAllowedToMoveUp	: BOOL;
	i_xAllowedToMoveDown: BOOL;
	i_xAlarmReset		: BOOL;
	
	// Hall Sensors
	i_xPin1HallSensorIn	: BOOL;
	i_xPin1HallSensorOut: BOOL;
	i_xPin2HallSensorIn	: BOOL;
	i_xPin2HallSensorOut: BOOL;	
	i_xPin3HallSensorIn	: BOOL;
	i_xPin3HallSensorOut: BOOL;	
	i_xPin4HallSensorIn	: BOOL;
	i_xPin4HallSensorOut: BOOL;
	
	i_xLightSensor1		: BOOL; // De eerste sensor die de pallet detecteerd
	i_xLightSensor2		: BOOL; // De tweede sensor die de pallet detecteerd
	
	i_xEndSwitch		: BOOL; // Check if the lift is down
	
	i_iServoEncoder		: INT;
	i_iDistanceSensor	: INT;
	i_iLayerHeight		: INT;	// Height of each layer
	i_iNumberOfLayers   : INT;  // Total number of layers
END_VAR
VAR_OUTPUT
	o_xMotor 			: BOOL; // Motor Lift
	o_xTargetPos		: INT;
	o_xErrorLift 		: BOOL;
	o_xAlarmLift 		: BOOL;
	
	o_xMagnetValve		: BOOL;
	o_xErrorImpaler 	: BOOL;
	o_xAlarmImpaler		: BOOL;
	
	o_xNewPalletPossible: BOOL;
	o_xPalletInPosition	: BOOL;
	o_eLiftPosition		: eLiftposition;
END_VAR
VAR
	iErrorCounter	: INT := 0; // Counts retries, after a few times errors will appear
	iHomePosition	: INT;
	iConveyorHeight	: INT;	// Standard height for grabbing or releasing pallet
	iImpaleHeight	: INT := iHomePosition + iConveyorHeight;
END_VAR

// Janno geeft door naar welke laag hij moet. Laag 0 = home, laag 1 = band, laag 2 = pallet op pallet, laag 3 = pallets hoog



//sim
IF i_iServoEncoder > o_xTargetPos AND o_xMotor  AND GVL.TimerShort.Q THEN
	i_iServoEncoder:=i_iServoEncoder-1;
ELSIF i_iServoEncoder < o_xTargetPos AND o_xMotor  AND GVL.TimerShort.Q THEN
	i_iServoEncoder:=i_iServoEncoder+1;
END_IF

IF i_iServoEncoder=0 THEN
	i_xEndSwitch:= TRUE;
ELSE 
	i_xEndSwitch:= FALSE;
END_IF
IF o_xMagnetValve AND GVL.TimerShort.Q THEN
	i_xPin1HallSensorIn:=FALSE;
	i_xPin2HallSensorIn:=FALSE;
	i_xPin3HallSensorIn:=FALSE;
	i_xPin4HallSensorIn:=FALSE;
	i_xPin1HallSensorOut:=TRUE;
	i_xPin2HallSensorOut:=TRUE;
	i_xPin3HallSensorOut:=TRUE;
	i_xPin4HallSensorOut:=TRUE;
ELSIF NOT o_xMagnetValve AND GVL.TimerShort.Q THEN
	i_xPin1HallSensorOut:=FALSE;
	i_xPin2HallSensorOut:=FALSE;
	i_xPin3HallSensorOut:=FALSE;
	i_xPin4HallSensorOut:=FALSE;
	i_xPin1HallSensorIn:=TRUE;
	i_xPin2HallSensorIn:=TRUE;
	i_xPin3HallSensorIn:=TRUE;
	i_xPin4HallSensorIn:=TRUE;

END_IF
//end sim
IF i_eLiftState= eLiftStates.Impale THEN
	o_xMagnetValve:=1;
ELSIF i_eLiftState= eLiftStates.Deimpale THEN
	o_xMagnetValve:=0;
ELSE
	o_xMagnetValve:=0;
END_IF
			IF i_eState=eSingleState.Aborted OR i_eState=eSingleState.Aborting THEN
				o_xMotor:=FALSE;
			ELSIF  i_iServoEncoder > o_xTargetPos OR i_iServoEncoder<o_xTargetPos  THEN
				o_xMotor:=TRUE;
			ELSIF i_iServoEncoder = o_xTargetPos THEN
				o_xMotor:=FALSE;
			END_IF
					CASE i_iMoveToLayer OF
						0 :
							o_xTargetPos:=0;
						1 :
							// Ga naar band hoogte
							o_xTargetPos:=4;
						2 : 
							// Ga naar stapelhoogte
							o_xTargetPos:=12;
						3 :
							//hoogte om pallet neer te zetten
							o_xTargetPos:=8;

					END_CASE

END_FUNCTION_BLOCK

// ---- POUs/FB_Blinking.TcPOU
FUNCTION_BLOCK FB_Blinking
VAR_IN_OUT
	io_xBlinking		: BOOL;
END_VAR
VAR
	tBlink     		: TON;       
    xBlink     		: BOOL;    
END_VAR

tBlink(IN := TRUE, PT := T#500MS);  

IF tBlink.Q THEN
    xBlink := NOT xBlink;     
    tBlink(IN := FALSE);        
ELSE
    tBlink(IN := TRUE);       
END_IF

io_xBlinking := xBlink;

END_FUNCTION_BLOCK
